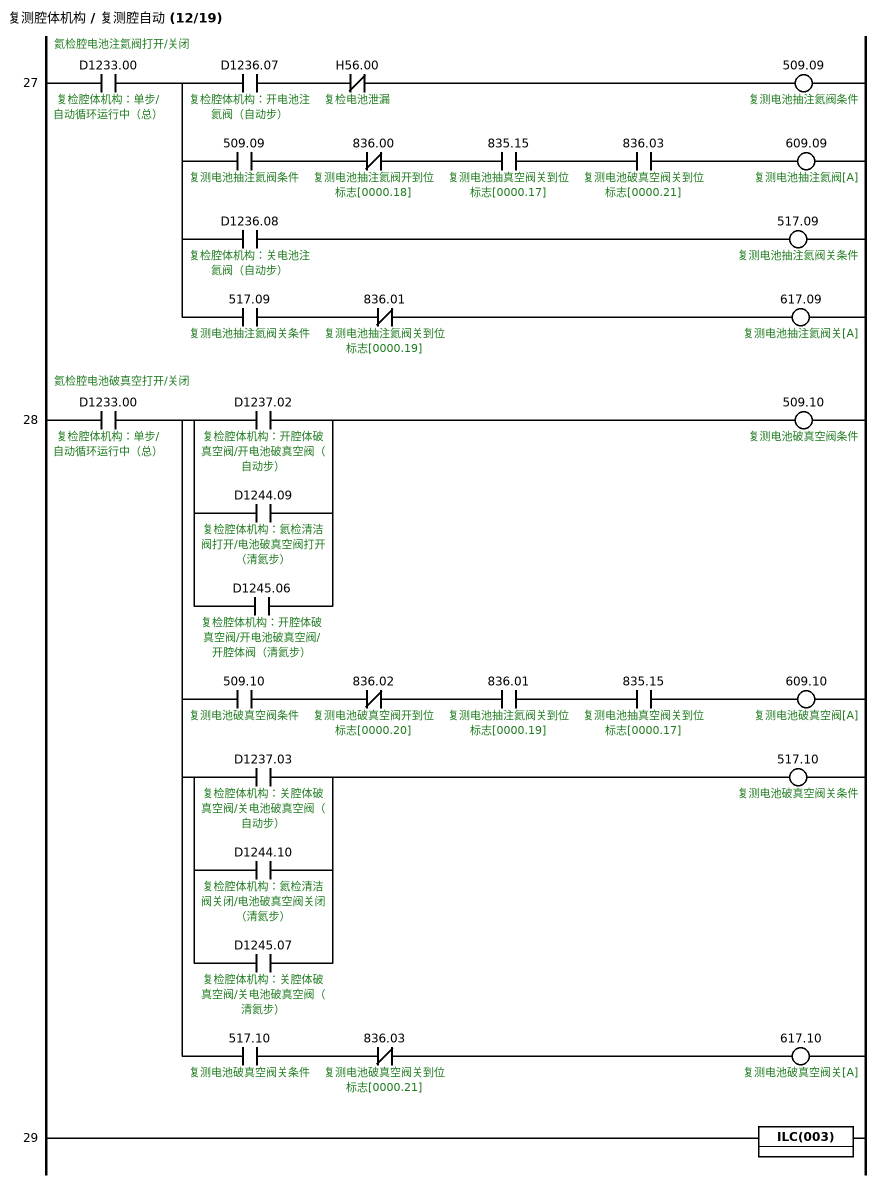
; [picture p600: 复测腔体机构 / 复测腔自动, rungs 27-29]
; rung 27: 氦检腔电池注氦阀打开/关闭
LD D1233.00  ; 复检腔体机构：单步/自动循环运行中（总）
OUT TR0
AND D1236.07  ; 复检腔体机构：开电池注氦阀（自动步）
ANDNOT H56.00  ; 复检电池泄漏
OUT 509.09  ; 复测电池抽注氦阀条件
LD TR0
AND 509.09  ; 复测电池抽注氦阀条件
ANDNOT 836.00  ; 复测电池抽注氦阀开到位标志[0000.18]
AND 835.15  ; 复测电池抽真空阀关到位标志[0000.17]
AND 836.03  ; 复测电池破真空阀关到位标志[0000.21]
OUT 609.09  ; 复测电池抽注氦阀[A]
LD TR0
AND D1236.08  ; 复检腔体机构：关电池注氦阀（自动步）
OUT 517.09  ; 复测电池抽注氦阀关条件
LD TR0
AND 517.09  ; 复测电池抽注氦阀关条件
ANDNOT 836.01  ; 复测电池抽注氦阀关到位标志[0000.19]
OUT 617.09  ; 复测电池抽注氦阀关[A]
; rung 28: 氦检腔电池破真空打开/关闭
LD D1233.00  ; 复检腔体机构：单步/自动循环运行中（总）
OUT TR0
LD D1237.02  ; 复检腔体机构：开腔体破真空阀/开电池破真空阀（自动步）
OR D1244.09  ; 复检腔体机构：氦检清洁阀打开/电池破真空阀打开（清氦步）
OR D1245.06  ; 复检腔体机构：开腔体破真空阀/开电池破真空阀/开腔体阀（清氦步）
ANDLD
OUT 509.10  ; 复测电池破真空阀条件
LD TR0
AND 509.10  ; 复测电池破真空阀条件
ANDNOT 836.02  ; 复测电池破真空阀开到位标志[0000.20]
AND 836.01  ; 复测电池抽注氦阀关到位标志[0000.19]
AND 835.15  ; 复测电池抽真空阀关到位标志[0000.17]
OUT 609.10  ; 复测电池破真空阀[A]
LD TR0
LD D1237.03  ; 复检腔体机构：关腔体破真空阀/关电池破真空阀（自动步）
OR D1244.10  ; 复检腔体机构：氦检清洁阀关闭/电池破真空阀关闭（清氦步）
OR D1245.07  ; 复检腔体机构：关腔体破真空阀/关电池破真空阀（清氦步）
ANDLD
OUT 517.10  ; 复测电池破真空阀关条件
LD TR0
AND 517.10  ; 复测电池破真空阀关条件
ANDNOT 836.03  ; 复测电池破真空阀关到位标志[0000.21]
OUT 617.10  ; 复测电池破真空阀关[A]
; rung 29
ILC(003)

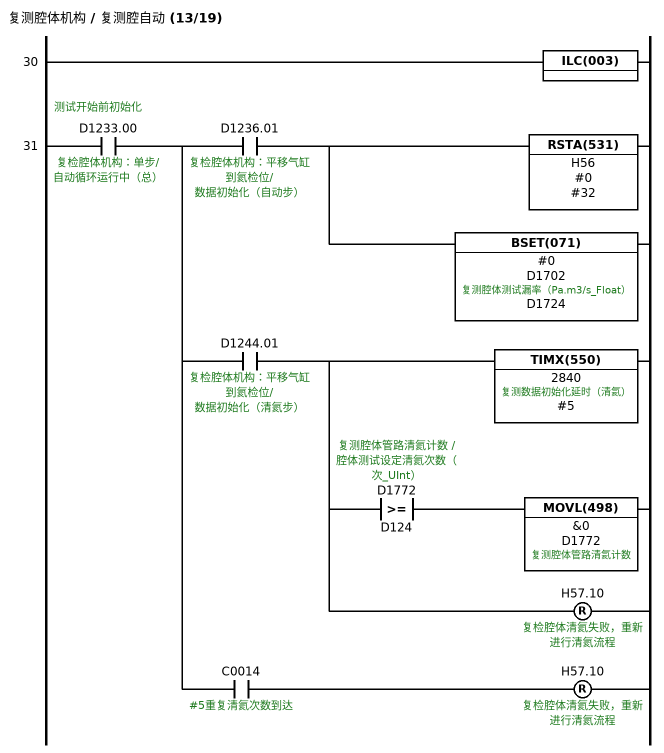
; rung 30
ILC(003)
; rung 31: 测试开始前初始化
LD D1233.00  ; 复检腔体机构：单步/自动循环运行中（总）
OUT TR0
AND D1236.01  ; 复检腔体机构：平移气缸到氦检位/数据初始化（自动步）
RSTA(531) H56 #0 #32
BSET(071) #0 D1702 D1724  ; 复测腔体测试漏率（Pa.m3/s_Float）
LD TR0
AND D1244.01  ; 复检腔体机构：平移气缸到氦检位/数据初始化（清氦步）
OUT TR1
TIMX(550) 2840 #5  ; 复测数据初始化延时（清氦）
AND>=(325) D1772 D124  ; 复测腔体管路清氦计数, 腔体测试设定清氦次数（次_UInt）
MOVL(498) &0 D1772  ; 复测腔体管路清氦计数
LD TR1
RSET H57.10  ; 复检腔体清氦失败，重新进行清氦流程
LD TR0
AND C0014  ; #5重复清氦次数到达
RSET H57.10  ; 复检腔体清氦失败，重新进行清氦流程

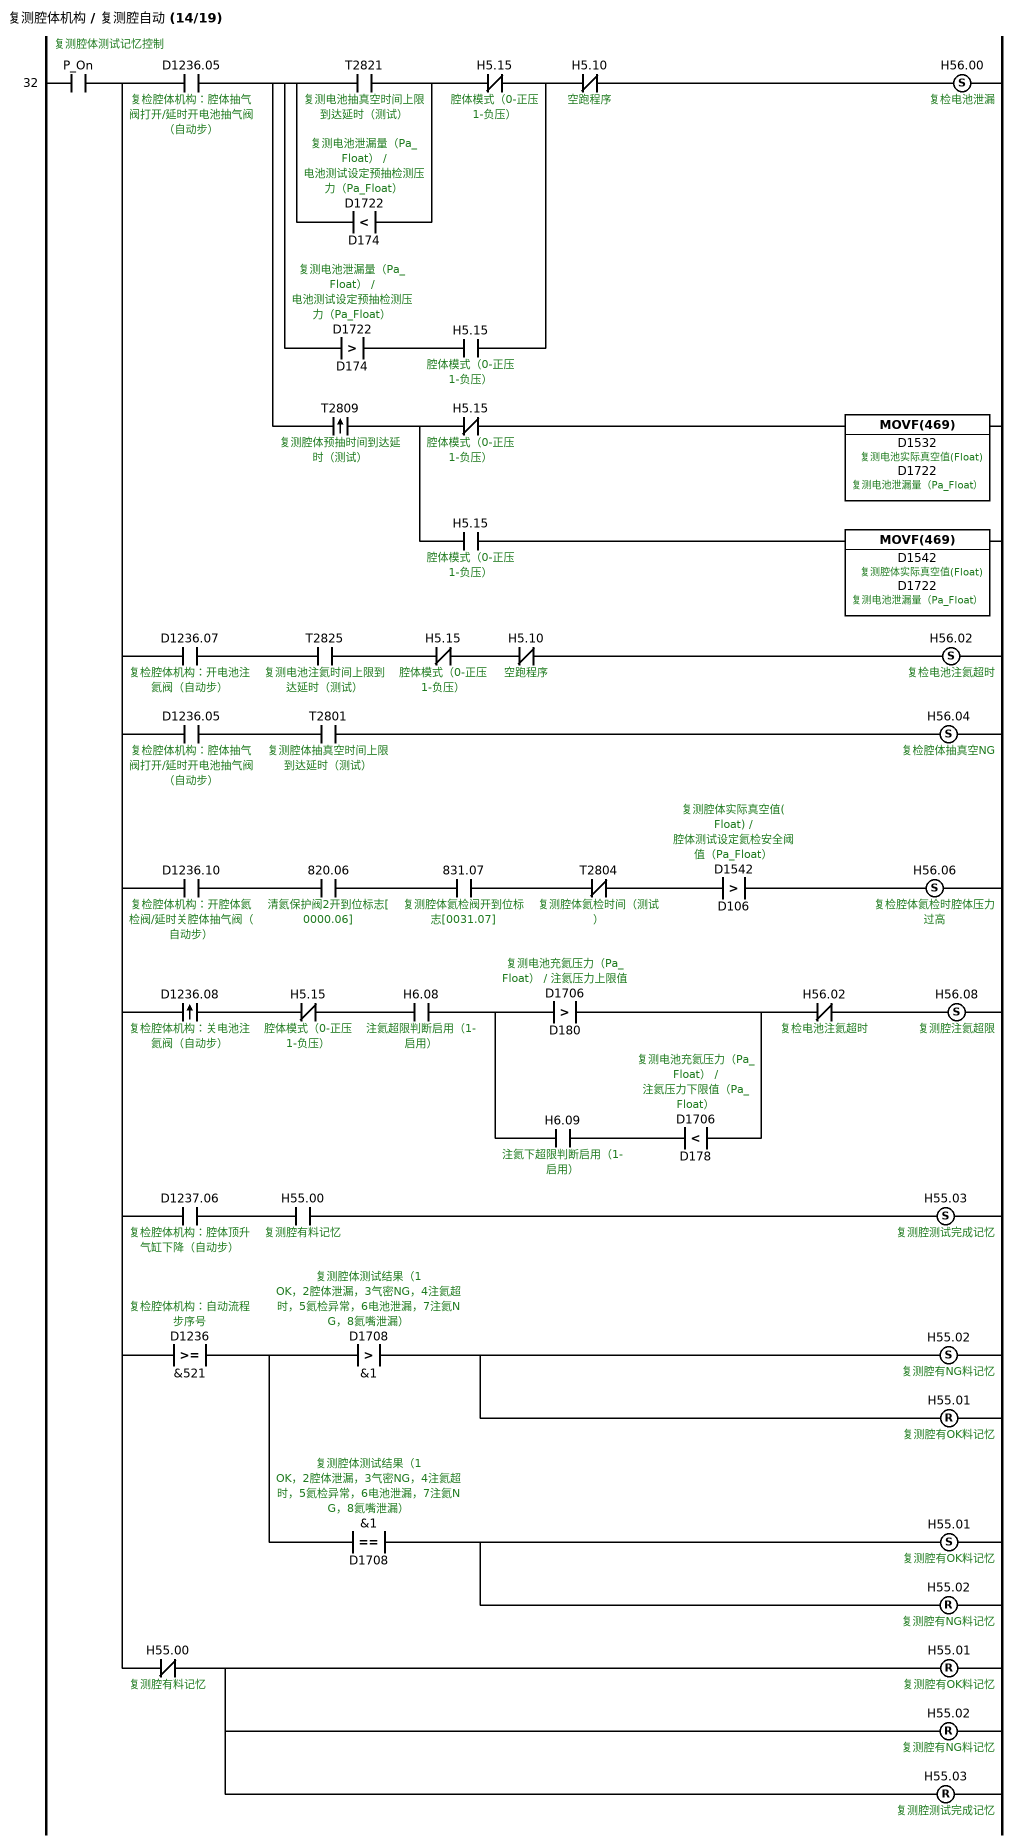
; rung 32: 复测腔体测试记忆控制
LD P_On
OUT TR0
AND D1236.05  ; 复检腔体机构：腔体抽气阀打开/延时开电池抽气阀（自动步）
OUT TR1
LD T2821  ; 复测电池抽真空时间上限到达延时（测试）
OR<F(331) D1722 D174  ; 复测电池泄漏量（Pa_Float）, 电池测试设定预抽检测压力（Pa_Float）
ANDNOT H5.15  ; 腔体模式（0-正压 1-负压）
LD>F(333) D1722 D174  ; 复测电池泄漏量（Pa_Float）, 电池测试设定预抽检测压力（Pa_Float）
AND H5.15  ; 腔体模式（0-正压 1-负压）
ORLD
ANDLD
ANDNOT H5.10  ; 空跑程序
SET H56.00  ; 复检电池泄漏
LD TR1
@AND T2809  ; 复测腔体预抽时间到达延时（测试）
OUT TR1
ANDNOT H5.15  ; 腔体模式（0-正压 1-负压）
MOVF(469) D1532 D1722  ; 复测电池实际真空值(Float), 复测电池泄漏量（Pa_Float）
LD TR1
AND H5.15  ; 腔体模式（0-正压 1-负压）
MOVF(469) D1542 D1722  ; 复测腔体实际真空值(Float), 复测电池泄漏量（Pa_Float）
LD TR0
AND D1236.07  ; 复检腔体机构：开电池注氦阀（自动步）
AND T2825  ; 复测电池注氦时间上限到达延时（测试）
ANDNOT H5.15  ; 腔体模式（0-正压 1-负压）
ANDNOT H5.10  ; 空跑程序
SET H56.02  ; 复检电池注氦超时
LD TR0
AND D1236.05  ; 复检腔体机构：腔体抽气阀打开/延时开电池抽气阀（自动步）
AND T2801  ; 复测腔体抽真空时间上限到达延时（测试）
SET H56.04  ; 复检腔体抽真空NG
LD TR0
AND D1236.10  ; 复检腔体机构：开腔体氦检阀/延时关腔体抽气阀（自动步）
AND 820.06  ; 清氦保护阀2开到位标志[0000.06]
AND 831.07  ; 复测腔体氦检阀开到位标志[0031.07]
ANDNOT T2804  ; 复测腔体氦检时间（测试）
AND>F(333) D1542 D106  ; 复测腔体实际真空值(Float), 腔体测试设定氦检安全阈值（Pa_Float）
SET H56.06  ; 复检腔体氦检时腔体压力过高
LD TR0
@AND D1236.08  ; 复检腔体机构：关电池注氦阀（自动步）
ANDNOT H5.15  ; 腔体模式（0-正压 1-负压）
AND H6.08  ; 注氦超限判断启用（1-启用）
LD>F(333) D1706 D180  ; 复测电池充氦压力（Pa_Float）, 注氦压力上限值
LD H6.09  ; 注氦下超限判断启用（1-启用）
AND<F(331) D1706 D178  ; 复测电池充氦压力（Pa_Float）, 注氦压力下限值（Pa_Float）
ORLD
ANDLD
ANDNOT H56.02  ; 复检电池注氦超时
SET H56.08  ; 复测腔注氦超限
LD TR0
AND D1237.06  ; 复检腔体机构：腔体顶升气缸下降（自动步）
AND H55.00  ; 复测腔有料记忆
SET H55.03  ; 复测腔测试完成记忆
LD TR0
AND>=L(326) D1236 &521  ; 复检腔体机构：自动流程步序号
OUT TR1
AND>(320) D1708 &1  ; 复测腔体测试结果（1 OK，2腔体泄漏，3气密NG，4注氦超时，5氦检异常，6电池泄漏，7注氦NG，8氦嘴泄漏）
SET H55.02  ; 复测腔有NG料记忆
RSET H55.01  ; 复测腔有OK料记忆
LD TR1
AND=(300) &1 D1708  ; 复测腔体测试结果（1 OK，2腔体泄漏，3气密NG，4注氦超时，5氦检异常，6电池泄漏，7注氦NG，8氦嘴泄漏）
SET H55.01  ; 复测腔有OK料记忆
RSET H55.02  ; 复测腔有NG料记忆
LD TR0
ANDNOT H55.00  ; 复测腔有料记忆
RSET H55.01  ; 复测腔有OK料记忆
RSET H55.02  ; 复测腔有NG料记忆
RSET H55.03  ; 复测腔测试完成记忆

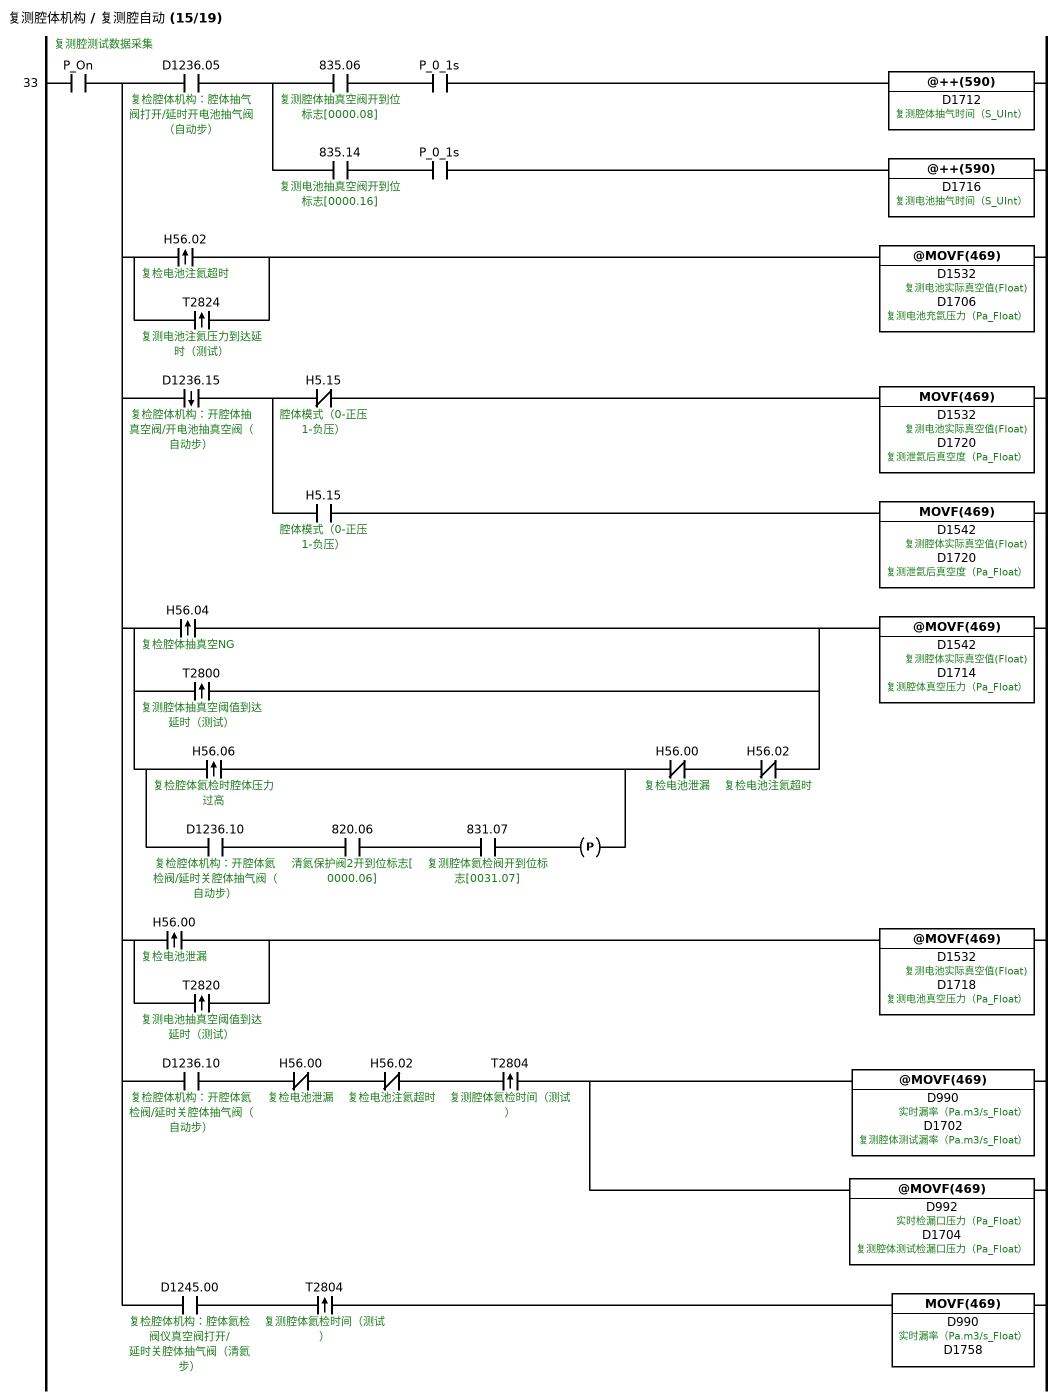
; rung 33: 复测腔测试数据采集
LD P_On
OUT TR0
AND D1236.05  ; 复检腔体机构：腔体抽气阀打开/延时开电池抽气阀（自动步）
OUT TR1
AND 835.06  ; 复测腔体抽真空阀开到位标志[0000.08]
AND P_0_1s
@++(590) D1712  ; 复测腔体抽气时间（S_UInt）
LD TR1
AND 835.14  ; 复测电池抽真空阀开到位标志[0000.16]
AND P_0_1s
@++(590) D1716  ; 复测电池抽气时间（S_UInt）
LD TR0
@LD H56.02  ; 复检电池注氦超时
@OR T2824  ; 复测电池注氦压力到达延时（测试）
ANDLD
@MOVF(469) D1532 D1706  ; 复测电池实际真空值(Float), 复测电池充氦压力（Pa_Float）
LD TR0
%AND D1236.15  ; 复检腔体机构：开腔体抽真空阀/开电池抽真空阀（自动步）
OUT TR1
ANDNOT H5.15  ; 腔体模式（0-正压 1-负压）
MOVF(469) D1532 D1720  ; 复测电池实际真空值(Float), 复测泄氦后真空度（Pa_Float）
LD TR1
AND H5.15  ; 腔体模式（0-正压 1-负压）
MOVF(469) D1542 D1720  ; 复测腔体实际真空值(Float), 复测泄氦后真空度（Pa_Float）
LD TR0
@LD H56.04  ; 复检腔体抽真空NG
@OR T2800  ; 复测腔体抽真空阈值到达延时（测试）
@LD H56.06  ; 复检腔体氦检时腔体压力过高
LD D1236.10  ; 复检腔体机构：开腔体氦检阀/延时关腔体抽气阀（自动步）
AND 820.06  ; 清氦保护阀2开到位标志[0000.06]
AND 831.07  ; 复测腔体氦检阀开到位标志[0031.07]
UP(521)
ORLD
ANDNOT H56.00  ; 复检电池泄漏
ANDNOT H56.02  ; 复检电池注氦超时
ORLD
ANDLD
@MOVF(469) D1542 D1714  ; 复测腔体实际真空值(Float), 复测腔体真空压力（Pa_Float）
LD TR0
@LD H56.00  ; 复检电池泄漏
@OR T2820  ; 复测电池抽真空阈值到达延时（测试）
ANDLD
@MOVF(469) D1532 D1718  ; 复测电池实际真空值(Float), 复测电池真空压力（Pa_Float）
LD TR0
AND D1236.10  ; 复检腔体机构：开腔体氦检阀/延时关腔体抽气阀（自动步）
ANDNOT H56.00  ; 复检电池泄漏
ANDNOT H56.02  ; 复检电池注氦超时
@AND T2804  ; 复测腔体氦检时间（测试）
@MOVF(469) D990 D1702  ; 实时漏率（Pa.m3/s_Float）, 复测腔体测试漏率（Pa.m3/s_Float）
@MOVF(469) D992 D1704  ; 实时检漏口压力（Pa_Float）, 复测腔体测试检漏口压力（Pa_Float）
LD TR0
AND D1245.00  ; 复检腔体机构：腔体氦检阀仪真空阀打开/延时关腔体抽气阀（清氦步）
@AND T2804  ; 复测腔体氦检时间（测试）
MOVF(469) D990 D1758  ; 实时漏率（Pa.m3/s_Float）

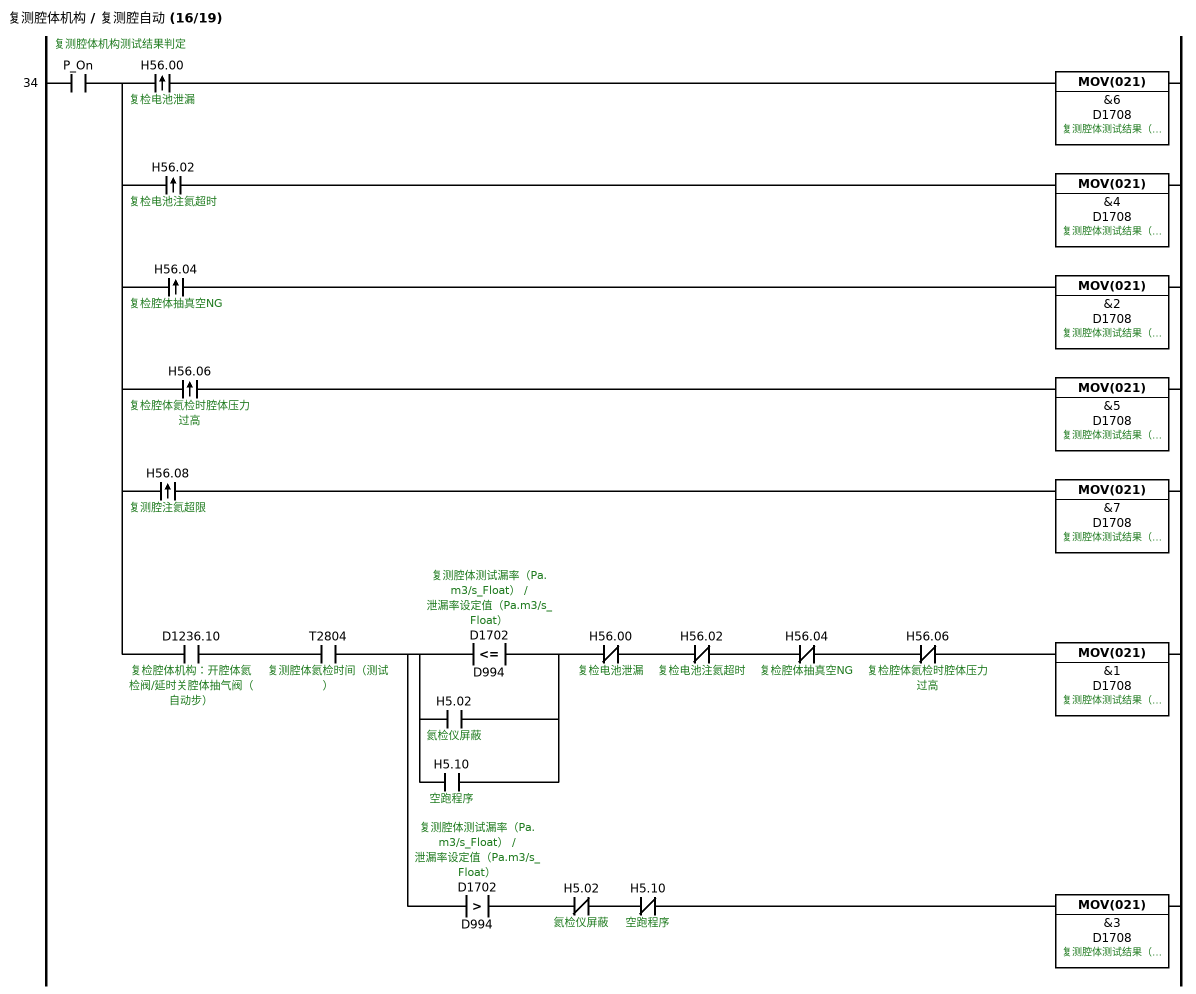
; rung 34: 复测腔体机构测试结果判定
LD P_On
OUT TR0
@AND H56.00  ; 复检电池泄漏
MOV(021) &6 D1708  ; 复测腔体测试结果（1 OK，2腔体泄漏，3气密NG，4注氦超时，5氦检异常，6电池泄漏，7注氦NG，8氦嘴泄漏）
LD TR0
@AND H56.02  ; 复检电池注氦超时
MOV(021) &4 D1708  ; 复测腔体测试结果（1 OK，2腔体泄漏，3气密NG，4注氦超时，5氦检异常，6电池泄漏，7注氦NG，8氦嘴泄漏）
LD TR0
@AND H56.04  ; 复检腔体抽真空NG
MOV(021) &2 D1708  ; 复测腔体测试结果（1 OK，2腔体泄漏，3气密NG，4注氦超时，5氦检异常，6电池泄漏，7注氦NG，8氦嘴泄漏）
LD TR0
@AND H56.06  ; 复检腔体氦检时腔体压力过高
MOV(021) &5 D1708  ; 复测腔体测试结果（1 OK，2腔体泄漏，3气密NG，4注氦超时，5氦检异常，6电池泄漏，7注氦NG，8氦嘴泄漏）
LD TR0
@AND H56.08  ; 复测腔注氦超限
MOV(021) &7 D1708  ; 复测腔体测试结果（1 OK，2腔体泄漏，3气密NG，4注氦超时，5氦检异常，6电池泄漏，7注氦NG，8氦嘴泄漏）
LD TR0
AND D1236.10  ; 复检腔体机构：开腔体氦检阀/延时关腔体抽气阀（自动步）
AND T2804  ; 复测腔体氦检时间（测试）
OUT TR0
LD<=F(332) D1702 D994  ; 复测腔体测试漏率（Pa.m3/s_Float）, 泄漏率设定值（Pa.m3/s_Float）
OR H5.02  ; 氦检仪屏蔽
OR H5.10  ; 空跑程序
ANDLD
ANDNOT H56.00  ; 复检电池泄漏
ANDNOT H56.02  ; 复检电池注氦超时
ANDNOT H56.04  ; 复检腔体抽真空NG
ANDNOT H56.06  ; 复检腔体氦检时腔体压力过高
MOV(021) &1 D1708  ; 复测腔体测试结果（1 OK，2腔体泄漏，3气密NG，4注氦超时，5氦检异常，6电池泄漏，7注氦NG，8氦嘴泄漏）
LD TR0
AND>F(333) D1702 D994  ; 复测腔体测试漏率（Pa.m3/s_Float）, 泄漏率设定值（Pa.m3/s_Float）
ANDNOT H5.02  ; 氦检仪屏蔽
ANDNOT H5.10  ; 空跑程序
MOV(021) &3 D1708  ; 复测腔体测试结果（1 OK，2腔体泄漏，3气密NG，4注氦超时，5氦检异常，6电池泄漏，7注氦NG，8氦嘴泄漏）

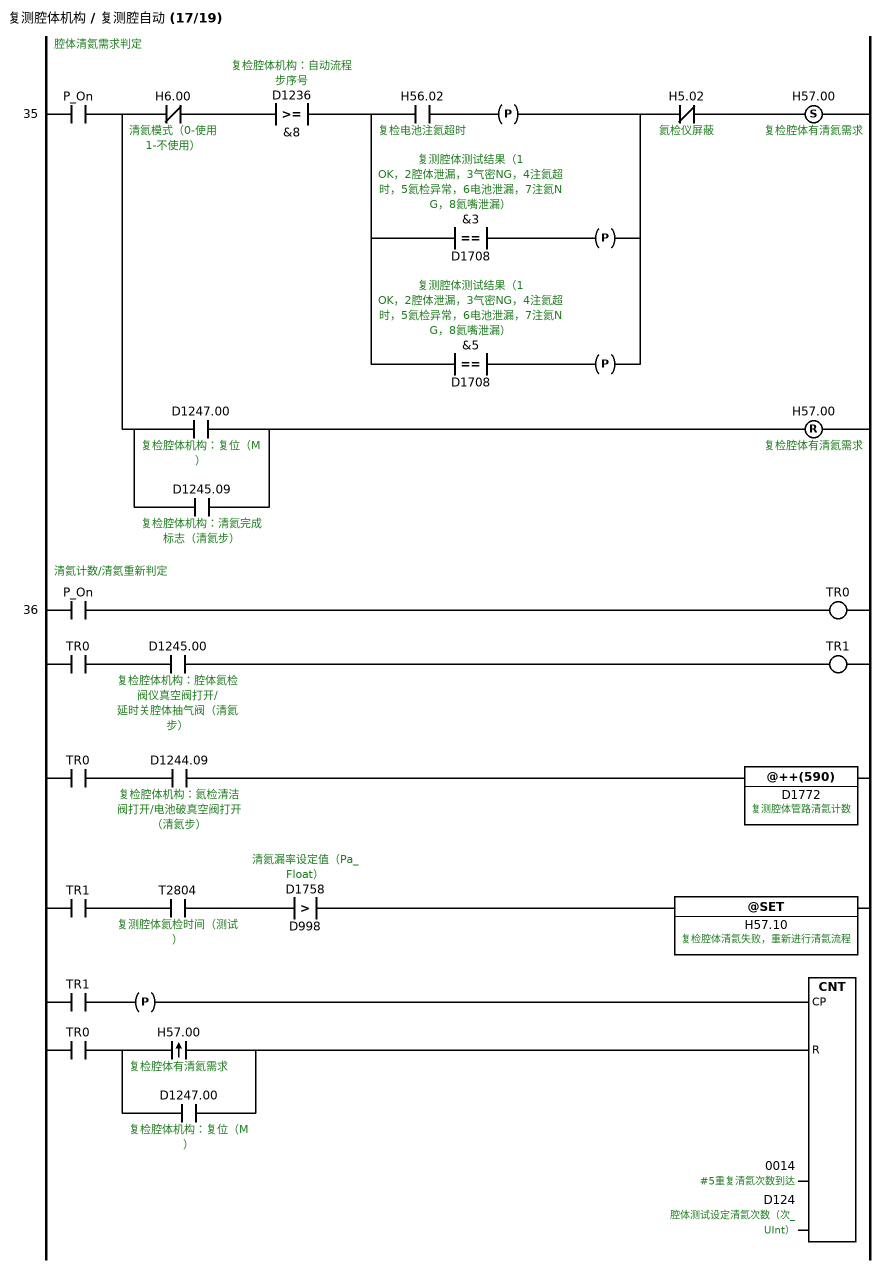
; rung 35: 腔体清氦需求判定
LD P_On
OUT TR0
ANDNOT H6.00  ; 清氦模式（0-使用 1-不使用）
AND>=L(326) D1236 &8  ; 复检腔体机构：自动流程步序号
LD H56.02  ; 复检电池注氦超时
UP(521)
LD=(300) &3 D1708  ; 复测腔体测试结果（1 OK，2腔体泄漏，3气密NG，4注氦超时，5氦检异常，6电池泄漏，7注氦NG，8氦嘴泄漏）
UP(521)
ORLD
LD=(300) &5 D1708  ; 复测腔体测试结果（1 OK，2腔体泄漏，3气密NG，4注氦超时，5氦检异常，6电池泄漏，7注氦NG，8氦嘴泄漏）
UP(521)
ORLD
ANDLD
ANDNOT H5.02  ; 氦检仪屏蔽
SET H57.00  ; 复检腔体有清氦需求
LD TR0
LD D1247.00  ; 复检腔体机构：复位（M）
OR D1245.09  ; 复检腔体机构：清氦完成标志（清氦步）
ANDLD
RSET H57.00  ; 复检腔体有清氦需求
; rung 36: 清氦计数/清氦重新判定
LD P_On
OUT TR0
AND D1244.09  ; 复检腔体机构：氦检清洁阀打开/电池破真空阀打开（清氦步）
@++(590) D1772  ; 复测腔体管路清氦计数
LD TR0
AND D1245.00  ; 复检腔体机构：腔体氦检阀仪真空阀打开/延时关腔体抽气阀（清氦步）
OUT TR1
AND T2804  ; 复测腔体氦检时间（测试）
AND>F(333) D1758 D998  ; 清氦漏率设定值（Pa_Float）
@SET H57.10  ; 复检腔体清氦失败，重新进行清氦流程
LD TR1
UP(521)
LD TR0
@LD H57.00  ; 复检腔体有清氦需求
OR D1247.00  ; 复检腔体机构：复位（M）
ANDLD
CNT 0014 D124  ; 腔体测试设定清氦次数（次_UInt）, #5重复清氦次数到达

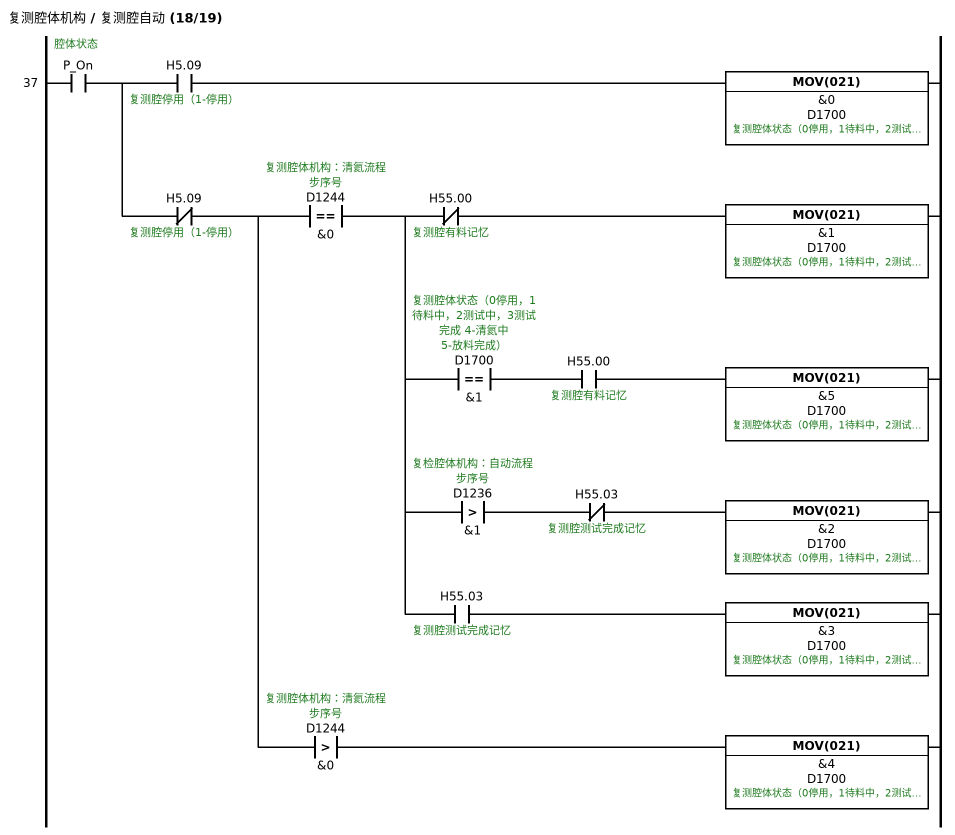
; rung 37: 腔体状态
LD P_On
OUT TR0
AND H5.09  ; 复测腔停用（1-停用）
MOV(021) &0 D1700  ; 复测腔体状态（0停用，1待料中，2测试中，3测试完成 4-清氦中  5-放料完成）
LD TR0
ANDNOT H5.09  ; 复测腔停用（1-停用）
OUT TR0
AND=L(301) D1244 &0  ; 复测腔体机构：清氦流程步序号
OUT TR1
ANDNOT H55.00  ; 复测腔有料记忆
MOV(021) &1 D1700  ; 复测腔体状态（0停用，1待料中，2测试中，3测试完成 4-清氦中  5-放料完成）
LD TR1
AND=(300) D1700 &1  ; 复测腔体状态（0停用，1待料中，2测试中，3测试完成 4-清氦中  5-放料完成）
AND H55.00  ; 复测腔有料记忆
MOV(021) &5 D1700  ; 复测腔体状态（0停用，1待料中，2测试中，3测试完成 4-清氦中  5-放料完成）
LD TR1
AND>L(321) D1236 &1  ; 复检腔体机构：自动流程步序号
ANDNOT H55.03  ; 复测腔测试完成记忆
MOV(021) &2 D1700  ; 复测腔体状态（0停用，1待料中，2测试中，3测试完成 4-清氦中  5-放料完成）
LD TR1
AND H55.03  ; 复测腔测试完成记忆
MOV(021) &3 D1700  ; 复测腔体状态（0停用，1待料中，2测试中，3测试完成 4-清氦中  5-放料完成）
LD TR0
AND>L(321) D1244 &0  ; 复测腔体机构：清氦流程步序号
MOV(021) &4 D1700  ; 复测腔体状态（0停用，1待料中，2测试中，3测试完成 4-清氦中  5-放料完成）

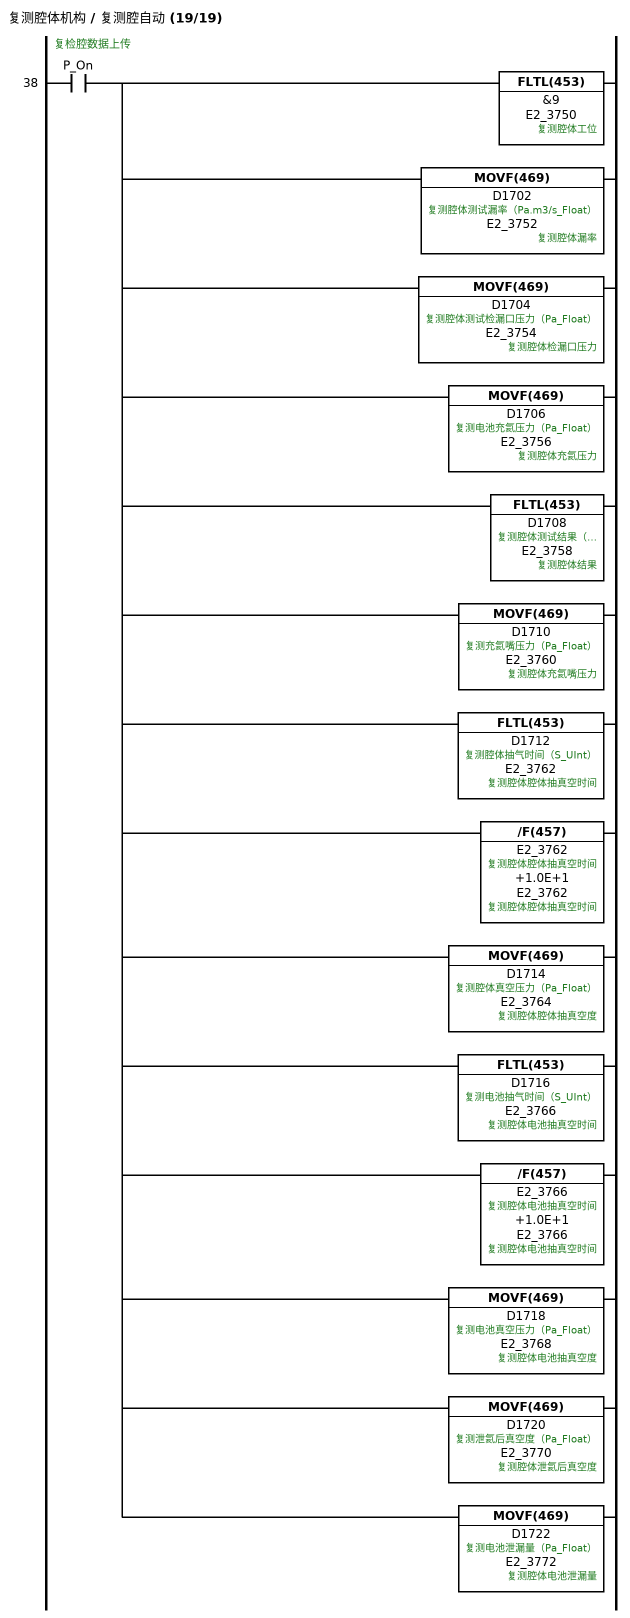
; rung 38: 复检腔数据上传
LD P_On
FLTL(453) &9 E2_3750  ; 复测腔体工位
MOVF(469) D1702 E2_3752  ; 复测腔体测试漏率（Pa.m3/s_Float）, 复测腔体漏率
MOVF(469) D1704 E2_3754  ; 复测腔体测试检漏口压力（Pa_Float）, 复测腔体检漏口压力
MOVF(469) D1706 E2_3756  ; 复测电池充氦压力（Pa_Float）, 复测腔体充氦压力
FLTL(453) D1708 E2_3758  ; 复测腔体测试结果（1 OK，2腔体泄漏，3气密NG，4注氦超时，5氦检异常，6电池泄漏，7注氦NG，8氦嘴泄漏）, 复测腔体结果
MOVF(469) D1710 E2_3760  ; 复测充氦嘴压力（Pa_Float）, 复测腔体充氦嘴压力
FLTL(453) D1712 E2_3762  ; 复测腔体抽气时间（S_UInt）, 复测腔体腔体抽真空时间
/F(457) E2_3762 +1.0E+1 E2_3762  ; 复测腔体腔体抽真空时间
MOVF(469) D1714 E2_3764  ; 复测腔体真空压力（Pa_Float）, 复测腔体腔体抽真空度
FLTL(453) D1716 E2_3766  ; 复测电池抽气时间（S_UInt）, 复测腔体电池抽真空时间
/F(457) E2_3766 +1.0E+1 E2_3766  ; 复测腔体电池抽真空时间
MOVF(469) D1718 E2_3768  ; 复测电池真空压力（Pa_Float）, 复测腔体电池抽真空度
MOVF(469) D1720 E2_3770  ; 复测泄氦后真空度（Pa_Float）, 复测腔体泄氦后真空度
MOVF(469) D1722 E2_3772  ; 复测电池泄漏量（Pa_Float）, 复测腔体电池泄漏量

### Section 复测腔手动

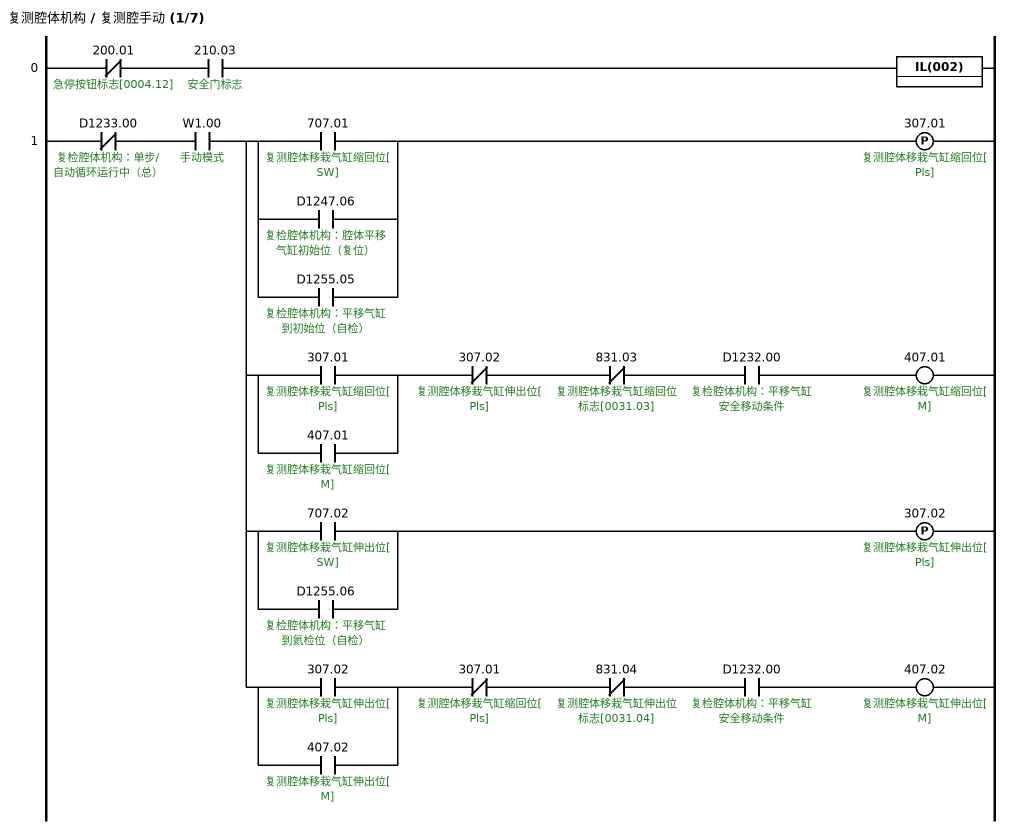
; rung 0
LDNOT 200.01  ; 急停按钮标志[0004.12]
AND 210.03  ; 安全门标志
IL(002)
; rung 1
LDNOT D1233.00  ; 复检腔体机构：单步/自动循环运行中（总）
AND W1.00  ; 手动模式
OUT TR0
LD 707.01  ; 复测腔体移栽气缸缩回位[SW]
OR D1247.06  ; 复检腔体机构：腔体平移气缸初始位（复位）
OR D1255.05  ; 复检腔体机构：平移气缸到初始位（自检）
ANDLD
DIFU(013) 307.01  ; 复测腔体移栽气缸缩回位[Pls]
LD TR0
LD 307.01  ; 复测腔体移栽气缸缩回位[Pls]
OR 407.01  ; 复测腔体移栽气缸缩回位[M]
ANDLD
ANDNOT 307.02  ; 复测腔体移栽气缸伸出位[Pls]
ANDNOT 831.03  ; 复测腔体移栽气缸缩回位标志[0031.03]
AND D1232.00  ; 复检腔体机构：平移气缸安全移动条件
OUT 407.01  ; 复测腔体移栽气缸缩回位[M]
LD TR0
LD 707.02  ; 复测腔体移栽气缸伸出位[SW]
OR D1255.06  ; 复检腔体机构：平移气缸到氦检位（自检）
ANDLD
DIFU(013) 307.02  ; 复测腔体移栽气缸伸出位[Pls]
LD TR0
LD 307.02  ; 复测腔体移栽气缸伸出位[Pls]
OR 407.02  ; 复测腔体移栽气缸伸出位[M]
ANDLD
ANDNOT 307.01  ; 复测腔体移栽气缸缩回位[Pls]
ANDNOT 831.04  ; 复测腔体移栽气缸伸出位标志[0031.04]
AND D1232.00  ; 复检腔体机构：平移气缸安全移动条件
OUT 407.02  ; 复测腔体移栽气缸伸出位[M]

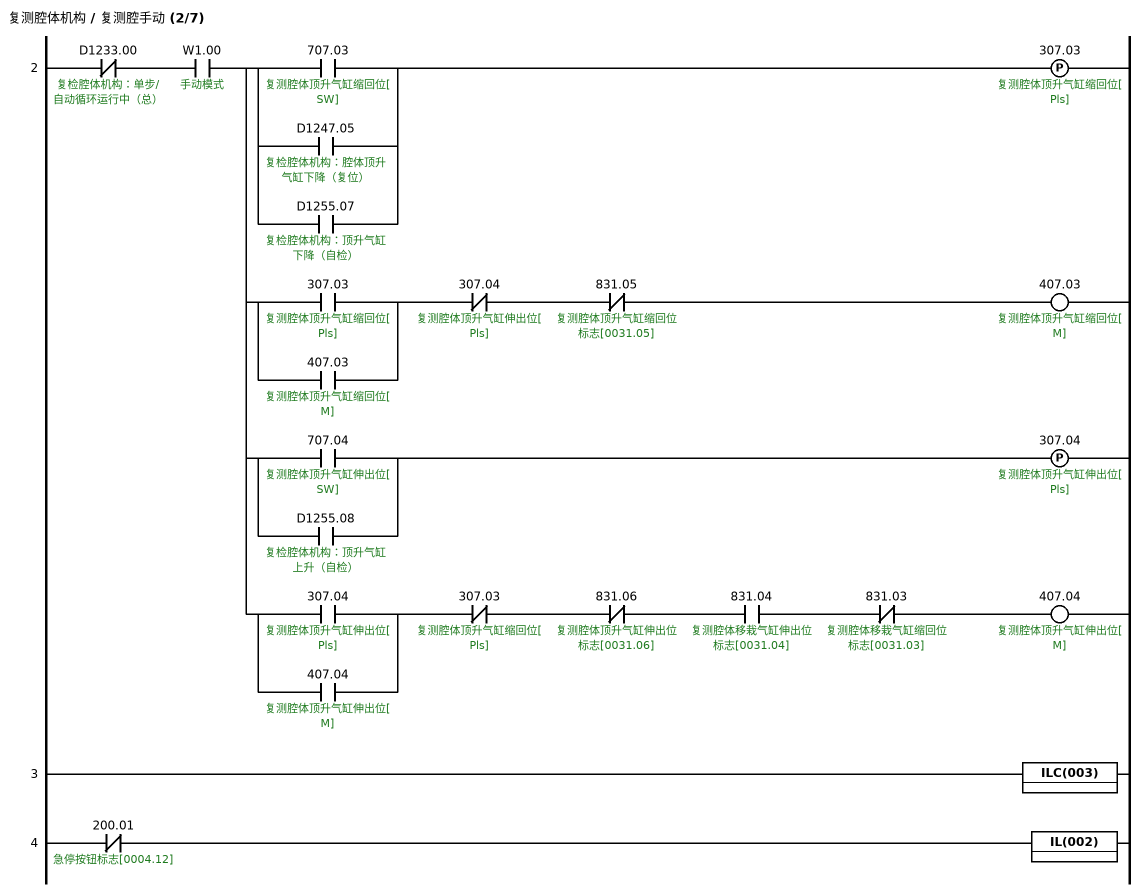
; rung 2
LDNOT D1233.00  ; 复检腔体机构：单步/自动循环运行中（总）
AND W1.00  ; 手动模式
OUT TR0
LD 707.03  ; 复测腔体顶升气缸缩回位[SW]
OR D1247.05  ; 复检腔体机构：腔体顶升气缸下降（复位）
OR D1255.07  ; 复检腔体机构：顶升气缸下降（自检）
ANDLD
DIFU(013) 307.03  ; 复测腔体顶升气缸缩回位[Pls]
LD TR0
LD 307.03  ; 复测腔体顶升气缸缩回位[Pls]
OR 407.03  ; 复测腔体顶升气缸缩回位[M]
ANDLD
ANDNOT 307.04  ; 复测腔体顶升气缸伸出位[Pls]
ANDNOT 831.05  ; 复测腔体顶升气缸缩回位标志[0031.05]
OUT 407.03  ; 复测腔体顶升气缸缩回位[M]
LD TR0
LD 707.04  ; 复测腔体顶升气缸伸出位[SW]
OR D1255.08  ; 复检腔体机构：顶升气缸上升（自检）
ANDLD
DIFU(013) 307.04  ; 复测腔体顶升气缸伸出位[Pls]
LD TR0
LD 307.04  ; 复测腔体顶升气缸伸出位[Pls]
OR 407.04  ; 复测腔体顶升气缸伸出位[M]
ANDLD
ANDNOT 307.03  ; 复测腔体顶升气缸缩回位[Pls]
ANDNOT 831.06  ; 复测腔体顶升气缸伸出位标志[0031.06]
AND 831.04  ; 复测腔体移栽气缸伸出位标志[0031.04]
ANDNOT 831.03  ; 复测腔体移栽气缸缩回位标志[0031.03]
OUT 407.04  ; 复测腔体顶升气缸伸出位[M]
; rung 3
ILC(003)
; rung 4
LDNOT 200.01  ; 急停按钮标志[0004.12]
IL(002)

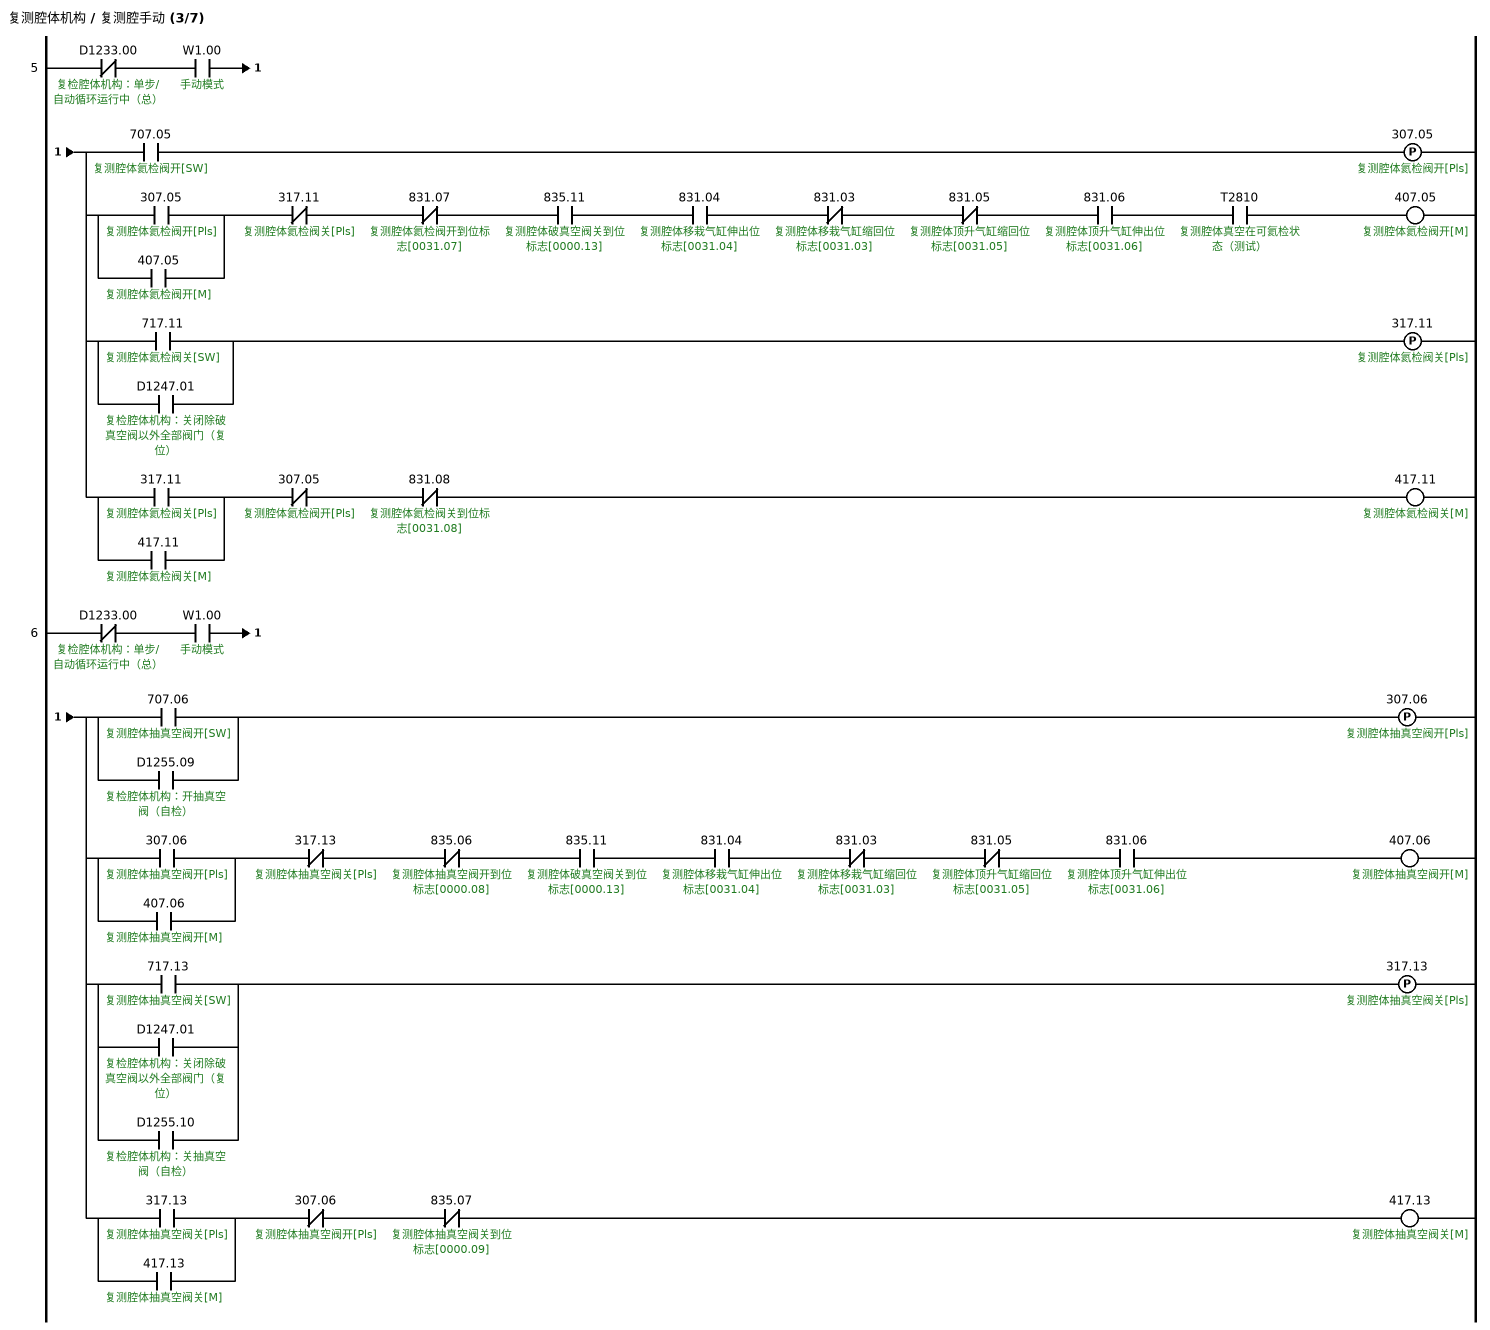
; rung 5
LDNOT D1233.00  ; 复检腔体机构：单步/自动循环运行中（总）
AND W1.00  ; 手动模式
OUT TR0
AND 707.05  ; 复测腔体氦检阀开[SW]
DIFU(013) 307.05  ; 复测腔体氦检阀开[Pls]
LD TR0
LD 307.05  ; 复测腔体氦检阀开[Pls]
OR 407.05  ; 复测腔体氦检阀开[M]
ANDLD
ANDNOT 317.11  ; 复测腔体氦检阀关[Pls]
ANDNOT 831.07  ; 复测腔体氦检阀开到位标志[0031.07]
AND 835.11  ; 复测腔体破真空阀关到位标志[0000.13]
AND 831.04  ; 复测腔体移栽气缸伸出位标志[0031.04]
ANDNOT 831.03  ; 复测腔体移栽气缸缩回位标志[0031.03]
ANDNOT 831.05  ; 复测腔体顶升气缸缩回位标志[0031.05]
AND 831.06  ; 复测腔体顶升气缸伸出位标志[0031.06]
AND T2810  ; 复测腔体真空在可氦检状态（测试）
OUT 407.05  ; 复测腔体氦检阀开[M]
LD TR0
LD 717.11  ; 复测腔体氦检阀关[SW]
OR D1247.01  ; 复检腔体机构：关闭除破真空阀以外全部阀门（复位）
ANDLD
DIFU(013) 317.11  ; 复测腔体氦检阀关[Pls]
LD TR0
LD 317.11  ; 复测腔体氦检阀关[Pls]
OR 417.11  ; 复测腔体氦检阀关[M]
ANDLD
ANDNOT 307.05  ; 复测腔体氦检阀开[Pls]
ANDNOT 831.08  ; 复测腔体氦检阀关到位标志[0031.08]
OUT 417.11  ; 复测腔体氦检阀关[M]
; rung 6
LDNOT D1233.00  ; 复检腔体机构：单步/自动循环运行中（总）
AND W1.00  ; 手动模式
OUT TR0
LD 707.06  ; 复测腔体抽真空阀开[SW]
OR D1255.09  ; 复检腔体机构：开抽真空阀（自检）
ANDLD
DIFU(013) 307.06  ; 复测腔体抽真空阀开[Pls]
LD TR0
LD 307.06  ; 复测腔体抽真空阀开[Pls]
OR 407.06  ; 复测腔体抽真空阀开[M]
ANDLD
ANDNOT 317.13  ; 复测腔体抽真空阀关[Pls]
ANDNOT 835.06  ; 复测腔体抽真空阀开到位标志[0000.08]
AND 835.11  ; 复测腔体破真空阀关到位标志[0000.13]
AND 831.04  ; 复测腔体移栽气缸伸出位标志[0031.04]
ANDNOT 831.03  ; 复测腔体移栽气缸缩回位标志[0031.03]
ANDNOT 831.05  ; 复测腔体顶升气缸缩回位标志[0031.05]
AND 831.06  ; 复测腔体顶升气缸伸出位标志[0031.06]
OUT 407.06  ; 复测腔体抽真空阀开[M]
LD TR0
LD 717.13  ; 复测腔体抽真空阀关[SW]
OR D1247.01  ; 复检腔体机构：关闭除破真空阀以外全部阀门（复位）
OR D1255.10  ; 复检腔体机构：关抽真空阀（自检）
ANDLD
DIFU(013) 317.13  ; 复测腔体抽真空阀关[Pls]
LD TR0
LD 317.13  ; 复测腔体抽真空阀关[Pls]
OR 417.13  ; 复测腔体抽真空阀关[M]
ANDLD
ANDNOT 307.06  ; 复测腔体抽真空阀开[Pls]
ANDNOT 835.07  ; 复测腔体抽真空阀关到位标志[0000.09]
OUT 417.13  ; 复测腔体抽真空阀关[M]

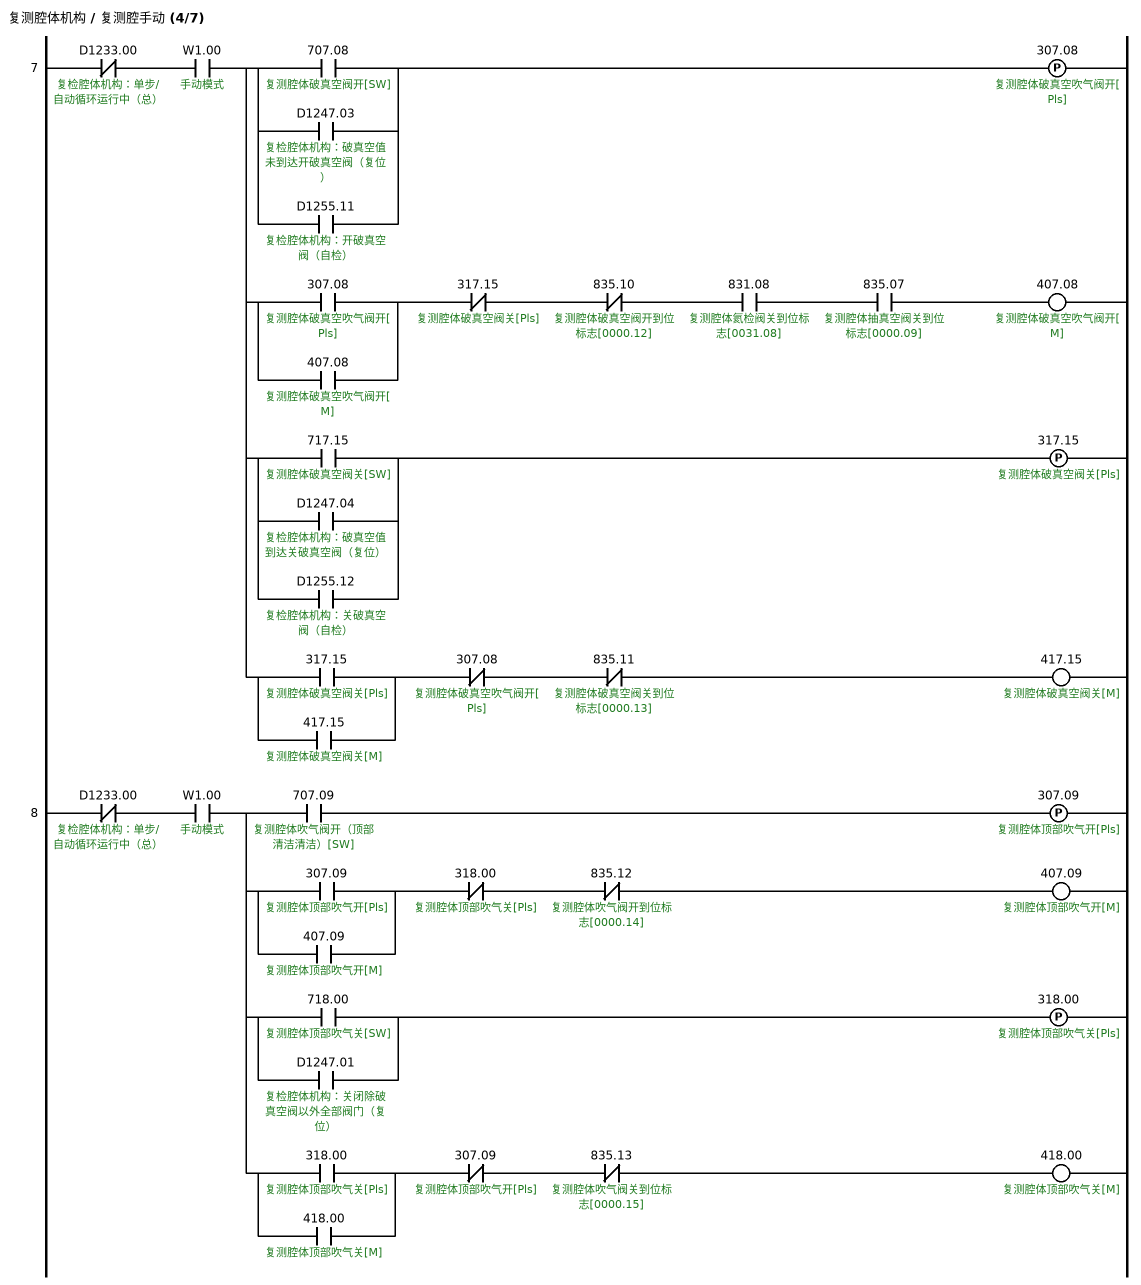
; rung 7
LDNOT D1233.00  ; 复检腔体机构：单步/自动循环运行中（总）
AND W1.00  ; 手动模式
OUT TR0
LD 707.08  ; 复测腔体破真空阀开[SW]
OR D1247.03  ; 复检腔体机构：破真空值未到达开破真空阀（复位）
OR D1255.11  ; 复检腔体机构：开破真空阀（自检）
ANDLD
DIFU(013) 307.08  ; 复测腔体破真空吹气阀开[Pls]
LD TR0
LD 307.08  ; 复测腔体破真空吹气阀开[Pls]
OR 407.08  ; 复测腔体破真空吹气阀开[M]
ANDLD
ANDNOT 317.15  ; 复测腔体破真空阀关[Pls]
ANDNOT 835.10  ; 复测腔体破真空阀开到位标志[0000.12]
AND 831.08  ; 复测腔体氦检阀关到位标志[0031.08]
AND 835.07  ; 复测腔体抽真空阀关到位标志[0000.09]
OUT 407.08  ; 复测腔体破真空吹气阀开[M]
LD TR0
LD 717.15  ; 复测腔体破真空阀关[SW]
OR D1247.04  ; 复检腔体机构：破真空值到达关破真空阀（复位）
OR D1255.12  ; 复检腔体机构：关破真空阀（自检）
ANDLD
DIFU(013) 317.15  ; 复测腔体破真空阀关[Pls]
LD TR0
LD 317.15  ; 复测腔体破真空阀关[Pls]
OR 417.15  ; 复测腔体破真空阀关[M]
ANDLD
ANDNOT 307.08  ; 复测腔体破真空吹气阀开[Pls]
ANDNOT 835.11  ; 复测腔体破真空阀关到位标志[0000.13]
OUT 417.15  ; 复测腔体破真空阀关[M]
; rung 8
LDNOT D1233.00  ; 复检腔体机构：单步/自动循环运行中（总）
AND W1.00  ; 手动模式
OUT TR0
AND 707.09  ; 复测腔体吹气阀开（顶部清洁清洁）[SW]
DIFU(013) 307.09  ; 复测腔体顶部吹气开[Pls]
LD TR0
LD 307.09  ; 复测腔体顶部吹气开[Pls]
OR 407.09  ; 复测腔体顶部吹气开[M]
ANDLD
ANDNOT 318.00  ; 复测腔体顶部吹气关[Pls]
ANDNOT 835.12  ; 复测腔体吹气阀开到位标志[0000.14]
OUT 407.09  ; 复测腔体顶部吹气开[M]
LD TR0
LD 718.00  ; 复测腔体顶部吹气关[SW]
OR D1247.01  ; 复检腔体机构：关闭除破真空阀以外全部阀门（复位）
ANDLD
DIFU(013) 318.00  ; 复测腔体顶部吹气关[Pls]
LD TR0
LD 318.00  ; 复测腔体顶部吹气关[Pls]
OR 418.00  ; 复测腔体顶部吹气关[M]
ANDLD
ANDNOT 307.09  ; 复测腔体顶部吹气开[Pls]
ANDNOT 835.13  ; 复测腔体吹气阀关到位标志[0000.15]
OUT 418.00  ; 复测腔体顶部吹气关[M]

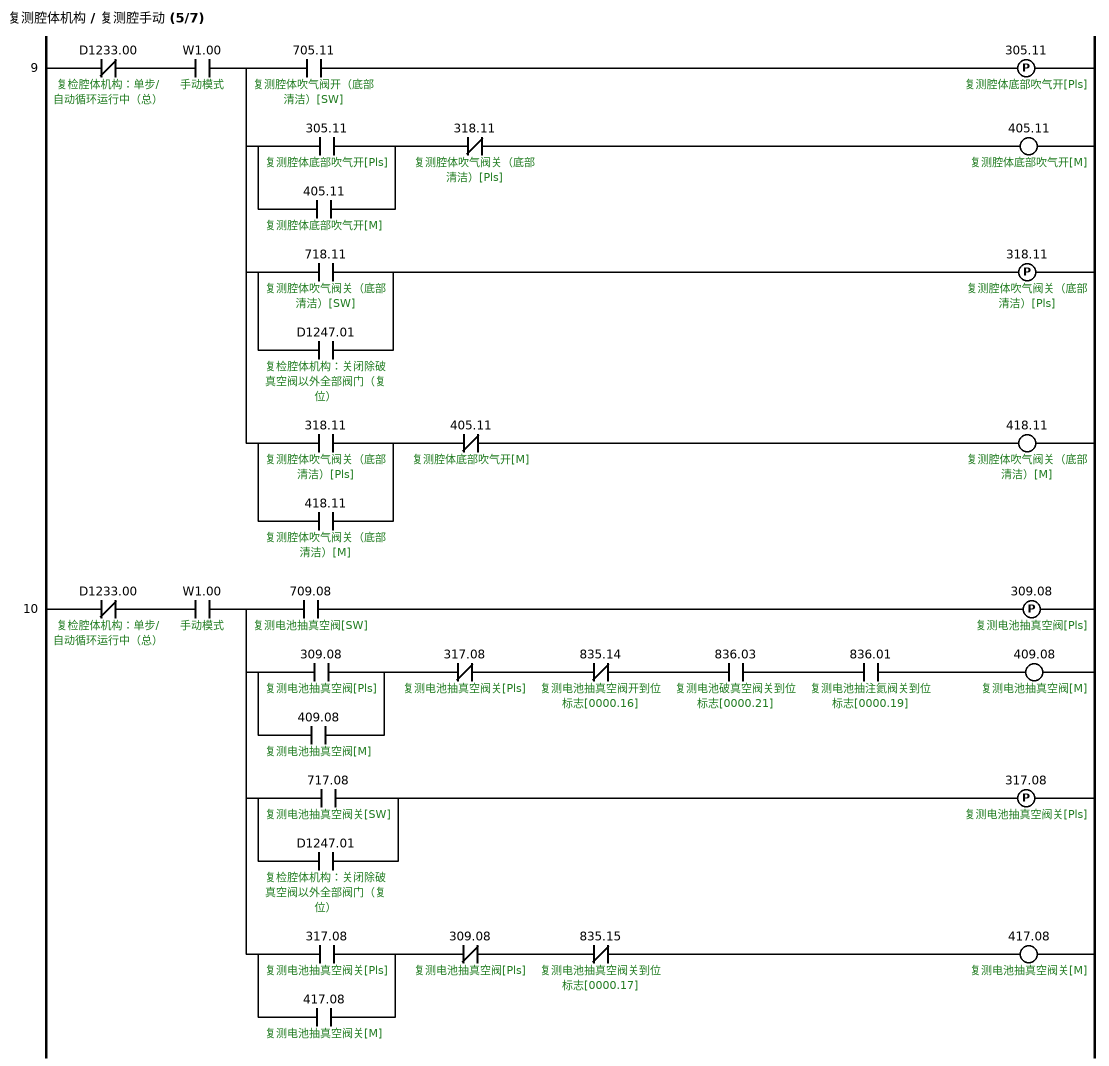
; rung 9
LDNOT D1233.00  ; 复检腔体机构：单步/自动循环运行中（总）
AND W1.00  ; 手动模式
OUT TR0
AND 705.11  ; 复测腔体吹气阀开（底部清洁）[SW]
DIFU(013) 305.11  ; 复测腔体底部吹气开[Pls]
LD TR0
LD 305.11  ; 复测腔体底部吹气开[Pls]
OR 405.11  ; 复测腔体底部吹气开[M]
ANDLD
ANDNOT 318.11  ; 复测腔体吹气阀关（底部清洁）[Pls]
OUT 405.11  ; 复测腔体底部吹气开[M]
LD TR0
LD 718.11  ; 复测腔体吹气阀关（底部清洁）[SW]
OR D1247.01  ; 复检腔体机构：关闭除破真空阀以外全部阀门（复位）
ANDLD
DIFU(013) 318.11  ; 复测腔体吹气阀关（底部清洁）[Pls]
LD TR0
LD 318.11  ; 复测腔体吹气阀关（底部清洁）[Pls]
OR 418.11  ; 复测腔体吹气阀关（底部清洁）[M]
ANDLD
ANDNOT 405.11  ; 复测腔体底部吹气开[M]
OUT 418.11  ; 复测腔体吹气阀关（底部清洁）[M]
; rung 10
LDNOT D1233.00  ; 复检腔体机构：单步/自动循环运行中（总）
AND W1.00  ; 手动模式
OUT TR0
AND 709.08  ; 复测电池抽真空阀[SW]
DIFU(013) 309.08  ; 复测电池抽真空阀[Pls]
LD TR0
LD 309.08  ; 复测电池抽真空阀[Pls]
OR 409.08  ; 复测电池抽真空阀[M]
ANDLD
ANDNOT 317.08  ; 复测电池抽真空阀关[Pls]
ANDNOT 835.14  ; 复测电池抽真空阀开到位标志[0000.16]
AND 836.03  ; 复测电池破真空阀关到位标志[0000.21]
AND 836.01  ; 复测电池抽注氦阀关到位标志[0000.19]
OUT 409.08  ; 复测电池抽真空阀[M]
LD TR0
LD 717.08  ; 复测电池抽真空阀关[SW]
OR D1247.01  ; 复检腔体机构：关闭除破真空阀以外全部阀门（复位）
ANDLD
DIFU(013) 317.08  ; 复测电池抽真空阀关[Pls]
LD TR0
LD 317.08  ; 复测电池抽真空阀关[Pls]
OR 417.08  ; 复测电池抽真空阀关[M]
ANDLD
ANDNOT 309.08  ; 复测电池抽真空阀[Pls]
ANDNOT 835.15  ; 复测电池抽真空阀关到位标志[0000.17]
OUT 417.08  ; 复测电池抽真空阀关[M]

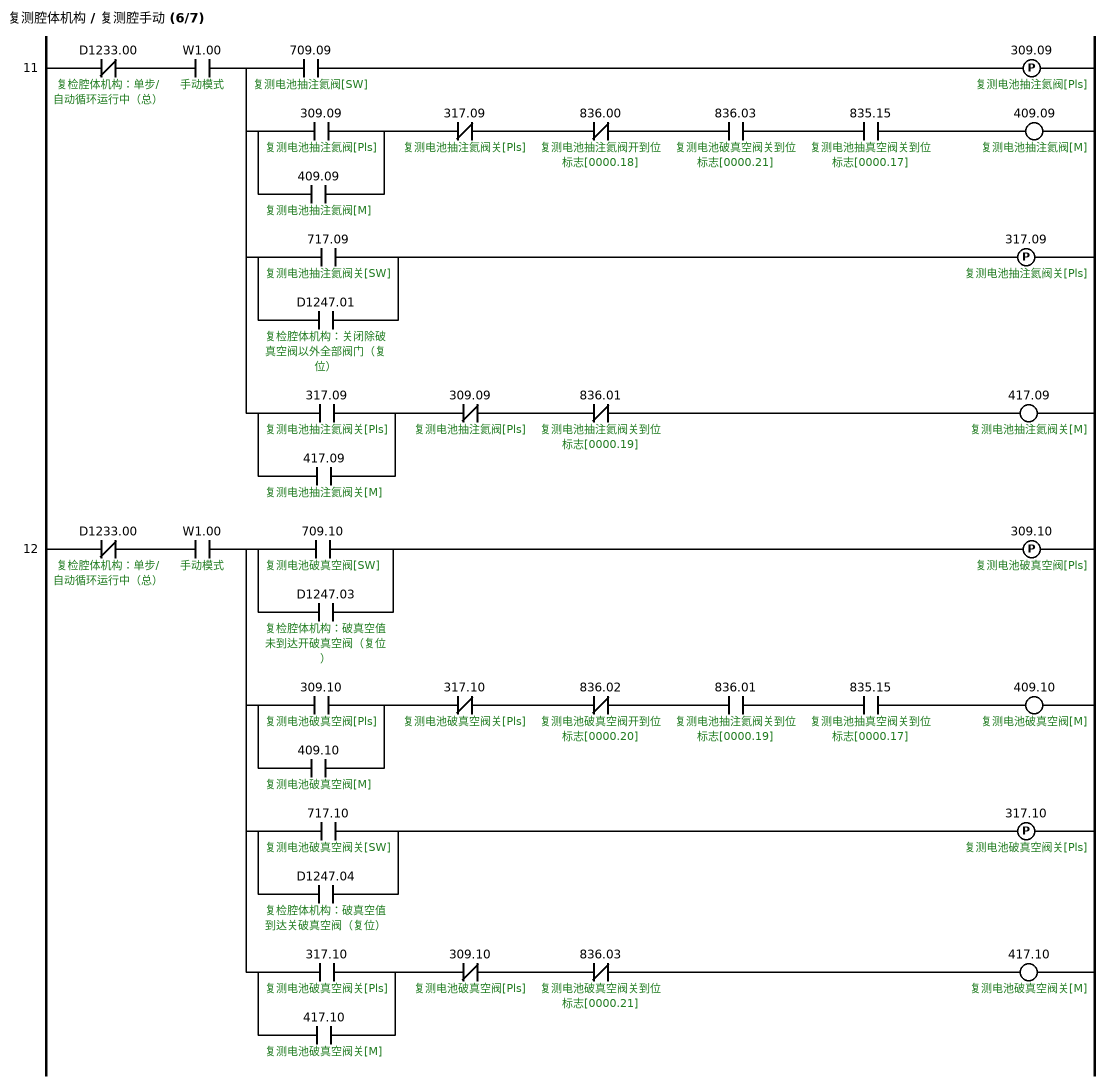
; rung 11
LDNOT D1233.00  ; 复检腔体机构：单步/自动循环运行中（总）
AND W1.00  ; 手动模式
OUT TR0
AND 709.09  ; 复测电池抽注氦阀[SW]
DIFU(013) 309.09  ; 复测电池抽注氦阀[Pls]
LD TR0
LD 309.09  ; 复测电池抽注氦阀[Pls]
OR 409.09  ; 复测电池抽注氦阀[M]
ANDLD
ANDNOT 317.09  ; 复测电池抽注氦阀关[Pls]
ANDNOT 836.00  ; 复测电池抽注氦阀开到位标志[0000.18]
AND 836.03  ; 复测电池破真空阀关到位标志[0000.21]
AND 835.15  ; 复测电池抽真空阀关到位标志[0000.17]
OUT 409.09  ; 复测电池抽注氦阀[M]
LD TR0
LD 717.09  ; 复测电池抽注氦阀关[SW]
OR D1247.01  ; 复检腔体机构：关闭除破真空阀以外全部阀门（复位）
ANDLD
DIFU(013) 317.09  ; 复测电池抽注氦阀关[Pls]
LD TR0
LD 317.09  ; 复测电池抽注氦阀关[Pls]
OR 417.09  ; 复测电池抽注氦阀关[M]
ANDLD
ANDNOT 309.09  ; 复测电池抽注氦阀[Pls]
ANDNOT 836.01  ; 复测电池抽注氦阀关到位标志[0000.19]
OUT 417.09  ; 复测电池抽注氦阀关[M]
; rung 12
LDNOT D1233.00  ; 复检腔体机构：单步/自动循环运行中（总）
AND W1.00  ; 手动模式
OUT TR0
LD 709.10  ; 复测电池破真空阀[SW]
OR D1247.03  ; 复检腔体机构：破真空值未到达开破真空阀（复位）
ANDLD
DIFU(013) 309.10  ; 复测电池破真空阀[Pls]
LD TR0
LD 309.10  ; 复测电池破真空阀[Pls]
OR 409.10  ; 复测电池破真空阀[M]
ANDLD
ANDNOT 317.10  ; 复测电池破真空阀关[Pls]
ANDNOT 836.02  ; 复测电池破真空阀开到位标志[0000.20]
AND 836.01  ; 复测电池抽注氦阀关到位标志[0000.19]
AND 835.15  ; 复测电池抽真空阀关到位标志[0000.17]
OUT 409.10  ; 复测电池破真空阀[M]
LD TR0
LD 717.10  ; 复测电池破真空阀关[SW]
OR D1247.04  ; 复检腔体机构：破真空值到达关破真空阀（复位）
ANDLD
DIFU(013) 317.10  ; 复测电池破真空阀关[Pls]
LD TR0
LD 317.10  ; 复测电池破真空阀关[Pls]
OR 417.10  ; 复测电池破真空阀关[M]
ANDLD
ANDNOT 309.10  ; 复测电池破真空阀[Pls]
ANDNOT 836.03  ; 复测电池破真空阀关到位标志[0000.21]
OUT 417.10  ; 复测电池破真空阀关[M]

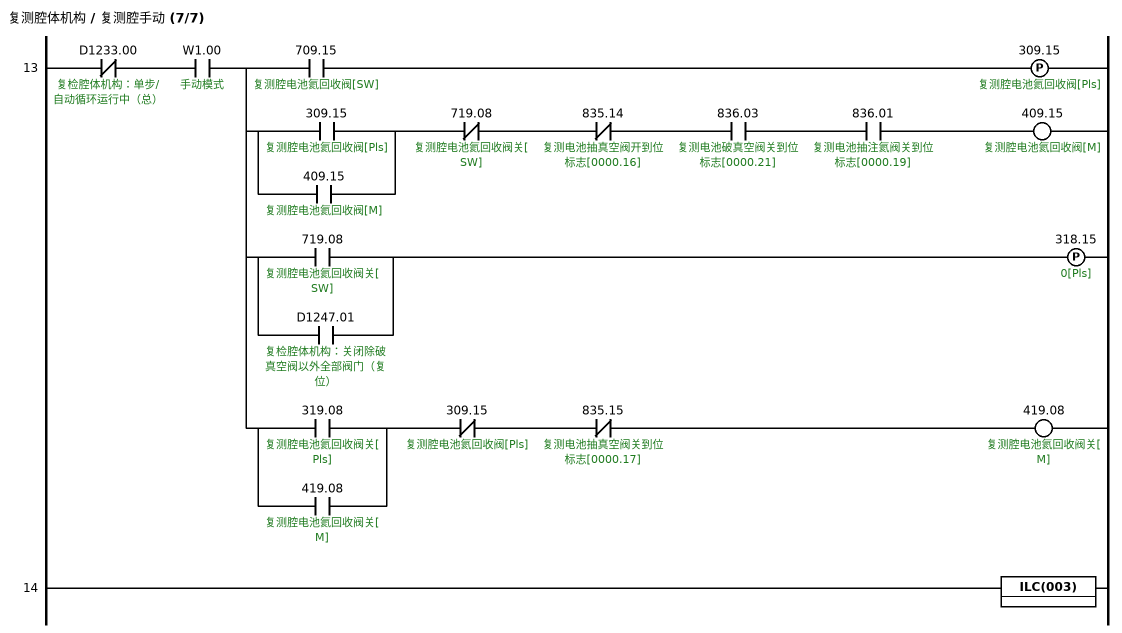
; rung 13
LDNOT D1233.00  ; 复检腔体机构：单步/自动循环运行中（总）
AND W1.00  ; 手动模式
OUT TR0
AND 709.15  ; 复测腔电池氦回收阀[SW]
DIFU(013) 309.15  ; 复测腔电池氦回收阀[Pls]
LD TR0
LD 309.15  ; 复测腔电池氦回收阀[Pls]
OR 409.15  ; 复测腔电池氦回收阀[M]
ANDLD
ANDNOT 719.08  ; 复测腔电池氦回收阀关[SW]
ANDNOT 835.14  ; 复测电池抽真空阀开到位标志[0000.16]
AND 836.03  ; 复测电池破真空阀关到位标志[0000.21]
AND 836.01  ; 复测电池抽注氦阀关到位标志[0000.19]
OUT 409.15  ; 复测腔电池氦回收阀[M]
LD TR0
LD 719.08  ; 复测腔电池氦回收阀关[SW]
OR D1247.01  ; 复检腔体机构：关闭除破真空阀以外全部阀门（复位）
ANDLD
DIFU(013) 318.15  ; 0[Pls]
LD TR0
LD 319.08  ; 复测腔电池氦回收阀关[Pls]
OR 419.08  ; 复测腔电池氦回收阀关[M]
ANDLD
ANDNOT 309.15  ; 复测腔电池氦回收阀[Pls]
ANDNOT 835.15  ; 复测电池抽真空阀关到位标志[0000.17]
OUT 419.08  ; 复测腔电池氦回收阀关[M]
; rung 14
ILC(003)

### Section 复检腔自检

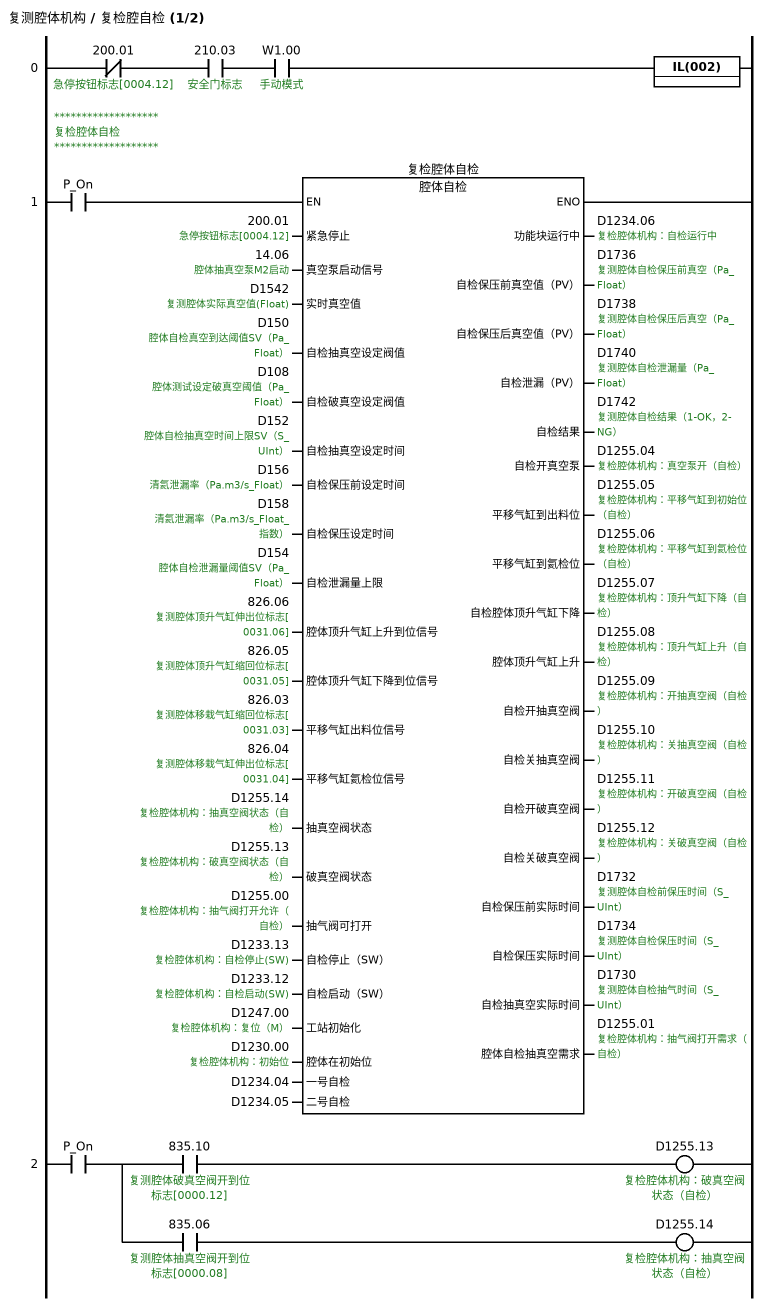
; rung 0
LDNOT 200.01  ; 急停按钮标志[0004.12]
AND 210.03  ; 安全门标志
AND W1.00  ; 手动模式
IL(002)
; rung 1: ******************* / 复检腔体自检 / *******************
LD P_On
CALL 复检腔体自检 : 腔体自检 (紧急停止 := 200.01, 真空泵启动信号 := 14.06, 实时真空值 := D1542, 自检抽真空设定阀值 := D150, 自检破真空设定阀值 := D108, 自检抽真空设定时间 := D152, 自检保压前设定时间 := D156, 自检保压设定时间 := D158, 自检泄漏量上限 := D154, 腔体顶升气缸上升到位信号 := 826.06, 腔体顶升气缸下降到位信号 := 826.05, 平移气缸出料位信号 := 826.03, 平移气缸氦检位信号 := 826.04, 抽真空阀状态 := D1255.14, 破真空阀状态 := D1255.13, 抽气阀可打开 := D1255.00, 自检停止（SW） := D1233.13, 自检启动（SW） := D1233.12, 工站初始化 := D1247.00, 腔体在初始位 := D1230.00, 一号自检 := D1234.04, 二号自检 := D1234.05, 功能块运行中 => D1234.06, 自检保压前真空值（PV） => D1736, 自检保压后真空值（PV） => D1738, 自检泄漏（PV） => D1740, 自检结果 => D1742, 自检开真空泵 => D1255.04, 平移气缸到出料位 => D1255.05, 平移气缸到氦检位 => D1255.06, 自检腔体顶升气缸下降 => D1255.07, 腔体顶升气缸上升 => D1255.08, 自检开抽真空阀 => D1255.09, 自检关抽真空阀 => D1255.10, 自检开破真空阀 => D1255.11, 自检关破真空阀 => D1255.12, 自检保压前实际时间 => D1732, 自检保压实际时间 => D1734, 自检抽真空实际时间 => D1730, 腔体自检抽真空需求 => D1255.01)  ; 急停按钮标志[0004.12], 腔体抽真空泵M2启动, 复测腔体实际真空值(Float), 腔体自检真空到达阈值SV（Pa_Float）, 腔体测试设定破真空阈值（Pa_Float）, 腔体自检抽真空时间上限SV（S_UInt）, 清氦泄漏率（Pa.m3/s_Float）, 清氦泄漏率（Pa.m3/s_Float_指数）, 腔体自检泄漏量阈值SV（Pa_Float）, 复测腔体顶升气缸伸出位标志[0031.06], 复测腔体顶升气缸缩回位标志[0031.05], 复测腔体移栽气缸缩回位标志[0031.03], 复测腔体移栽气缸伸出位标志[0031.04], 复检腔体机构：抽真空阀状态（自检）, 复检腔体机构：破真空阀状态（自检）, 复检腔体机构：抽气阀打开允许（自检）, 复检腔体机构：自检停止(SW), 复检腔体机构：自检启动(SW), 复检腔体机构：复位（M）, 复检腔体机构：初始位, 复检腔体机构：自检运行中, 复测腔体自检保压前真空（Pa_Float）, 复测腔体自检保压后真空（Pa_Float）, 复测腔体自检泄漏量（Pa_Float）, 复测腔体自检结果（1-OK，2-NG）, 复检腔体机构：真空泵开（自检）, 复检腔体机构：平移气缸到初始位（自检）, 复检腔体机构：平移气缸到氦检位（自检）, 复检腔体机构：顶升气缸下降（自检）, 复检腔体机构：顶升气缸上升（自检）, 复检腔体机构：开抽真空阀（自检）, 复检腔体机构：关抽真空阀（自检）, 复检腔体机构：开破真空阀（自检）, 复检腔体机构：关破真空阀（自检）, 复测腔体自检前保压时间（S_UInt）, 复测腔体自检保压时间（S_UInt）, 复测腔体自检抽气时间（S_UInt）, 复检腔体机构：抽气阀打开需求（自检）
; rung 2
LD P_On
OUT TR0
AND 835.10  ; 复测腔体破真空阀开到位标志[0000.12]
OUT D1255.13  ; 复检腔体机构：破真空阀状态（自检）
LD TR0
AND 835.06  ; 复测腔体抽真空阀开到位标志[0000.08]
OUT D1255.14  ; 复检腔体机构：抽真空阀状态（自检）

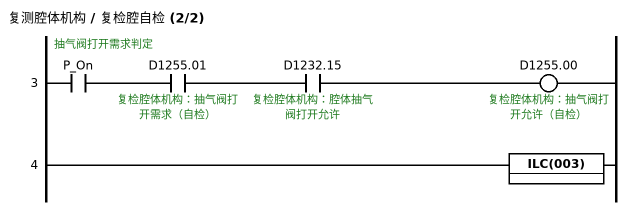
; rung 3: 抽气阀打开需求判定
LD P_On
AND D1255.01  ; 复检腔体机构：抽气阀打开需求（自检）
AND D1232.15  ; 复检腔体机构：腔体抽气阀打开允许
OUT D1255.00  ; 复检腔体机构：抽气阀打开允许（自检）
; rung 4
ILC(003)

### Section 工站复位

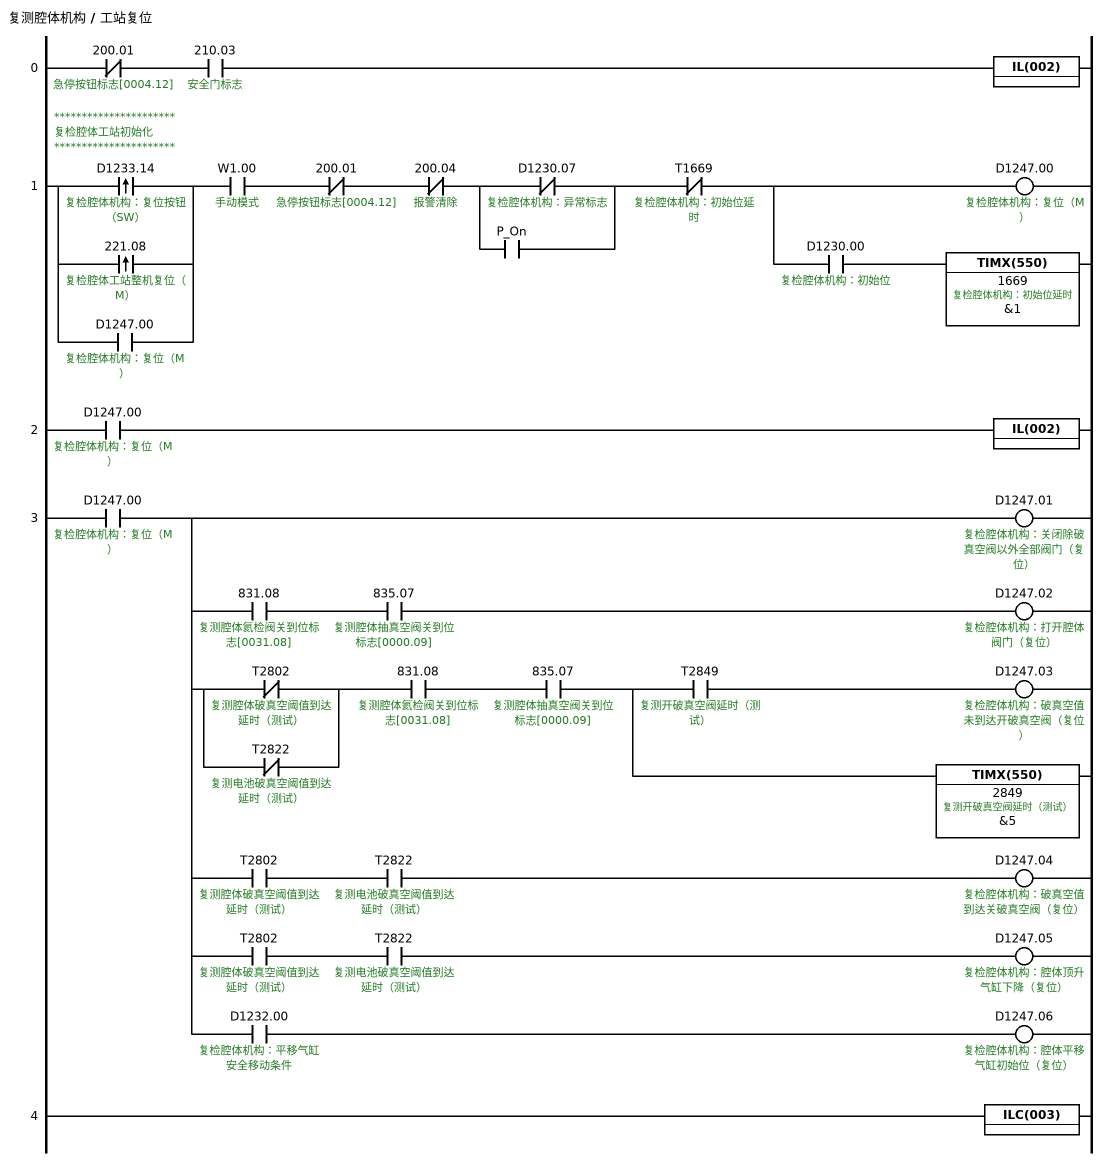
; rung 0
LDNOT 200.01  ; 急停按钮标志[0004.12]
AND 210.03  ; 安全门标志
IL(002)
; rung 1: ********************** / 复检腔体工站初始化 / **********************
@LD D1233.14  ; 复检腔体机构：复位按钮（SW）
@OR 221.08  ; 复检腔体工站整机复位（M）
OR D1247.00  ; 复检腔体机构：复位（M）
AND W1.00  ; 手动模式
ANDNOT 200.01  ; 急停按钮标志[0004.12]
ANDNOT 200.04  ; 报警清除
LDNOT D1230.07  ; 复检腔体机构：异常标志
OR P_On
ANDLD
ANDNOT T1669  ; 复检腔体机构：初始位延时
OUT D1247.00  ; 复检腔体机构：复位（M）
AND D1230.00  ; 复检腔体机构：初始位
TIMX(550) 1669 &1  ; 复检腔体机构：初始位延时
; rung 2
LD D1247.00  ; 复检腔体机构：复位（M）
IL(002)
; rung 3
LD D1247.00  ; 复检腔体机构：复位（M）
OUT TR0
OUT D1247.01  ; 复检腔体机构：关闭除破真空阀以外全部阀门（复位）
AND 831.08  ; 复测腔体氦检阀关到位标志[0031.08]
AND 835.07  ; 复测腔体抽真空阀关到位标志[0000.09]
OUT D1247.02  ; 复检腔体机构：打开腔体阀门（复位）
LD TR0
LDNOT T2802  ; 复测腔体破真空阈值到达延时（测试）
ORNOT T2822  ; 复测电池破真空阈值到达延时（测试）
ANDLD
AND 831.08  ; 复测腔体氦检阀关到位标志[0031.08]
AND 835.07  ; 复测腔体抽真空阀关到位标志[0000.09]
OUT TR1
AND T2849  ; 复测开破真空阀延时（测试）
OUT D1247.03  ; 复检腔体机构：破真空值未到达开破真空阀（复位）
LD TR1
TIMX(550) 2849 &5  ; 复测开破真空阀延时（测试）
LD TR0
AND T2802  ; 复测腔体破真空阈值到达延时（测试）
AND T2822  ; 复测电池破真空阈值到达延时（测试）
OUT D1247.04  ; 复检腔体机构：破真空值到达关破真空阀（复位）
LD TR0
AND T2802  ; 复测腔体破真空阈值到达延时（测试）
AND T2822  ; 复测电池破真空阈值到达延时（测试）
OUT D1247.05  ; 复检腔体机构：腔体顶升气缸下降（复位）
LD TR0
AND D1232.00  ; 复检腔体机构：平移气缸安全移动条件
OUT D1247.06  ; 复检腔体机构：腔体平移气缸初始位（复位）
; rung 4
ILC(003)

### Section 指示灯

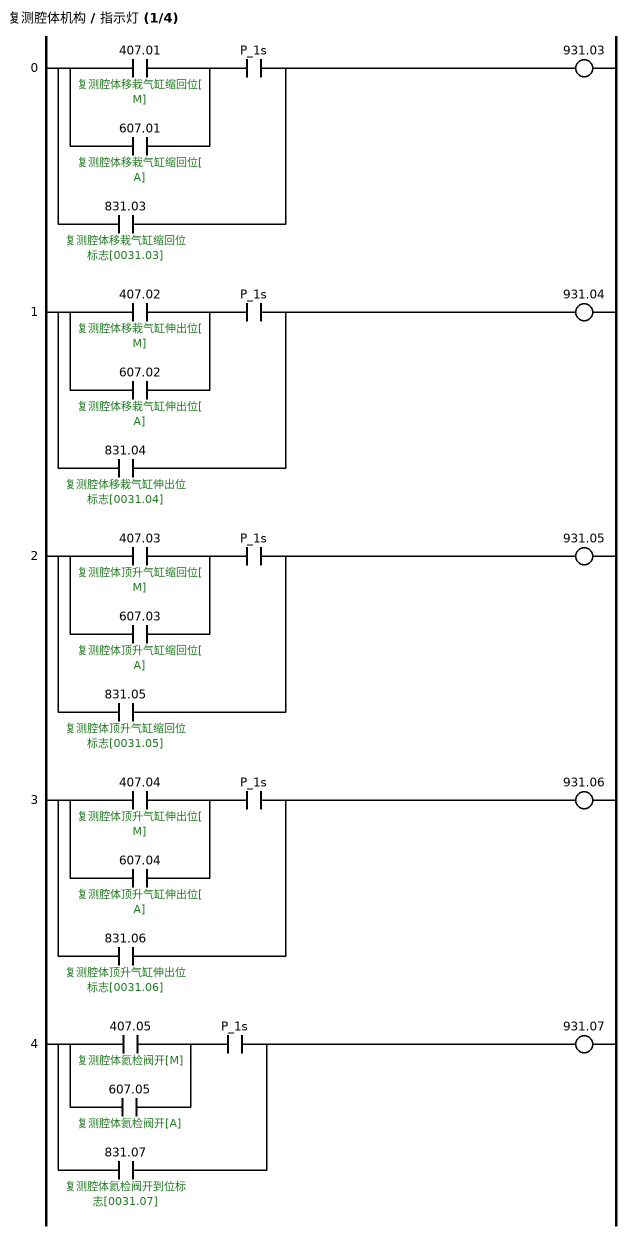
; rung 0
LD 407.01  ; 复测腔体移栽气缸缩回位[M]
OR 607.01  ; 复测腔体移栽气缸缩回位[A]
AND P_1s
OR 831.03  ; 复测腔体移栽气缸缩回位标志[0031.03]
OUT 931.03
; rung 1
LD 407.02  ; 复测腔体移栽气缸伸出位[M]
OR 607.02  ; 复测腔体移栽气缸伸出位[A]
AND P_1s
OR 831.04  ; 复测腔体移栽气缸伸出位标志[0031.04]
OUT 931.04
; rung 2
LD 407.03  ; 复测腔体顶升气缸缩回位[M]
OR 607.03  ; 复测腔体顶升气缸缩回位[A]
AND P_1s
OR 831.05  ; 复测腔体顶升气缸缩回位标志[0031.05]
OUT 931.05
; rung 3
LD 407.04  ; 复测腔体顶升气缸伸出位[M]
OR 607.04  ; 复测腔体顶升气缸伸出位[A]
AND P_1s
OR 831.06  ; 复测腔体顶升气缸伸出位标志[0031.06]
OUT 931.06
; rung 4
LD 407.05  ; 复测腔体氦检阀开[M]
OR 607.05  ; 复测腔体氦检阀开[A]
AND P_1s
OR 831.07  ; 复测腔体氦检阀开到位标志[0031.07]
OUT 931.07

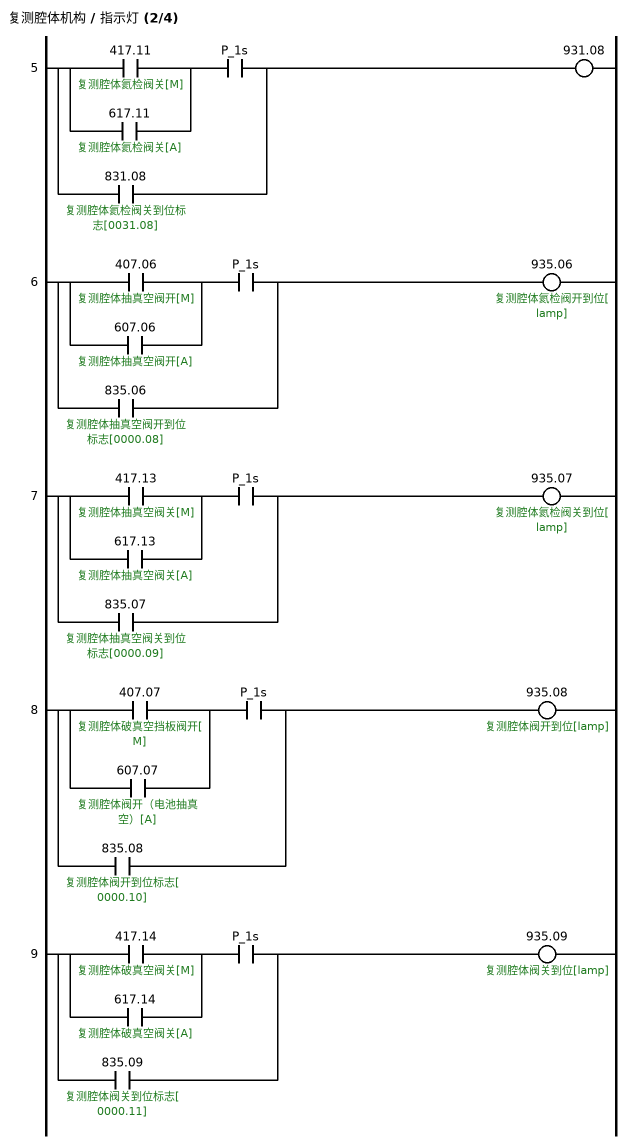
; rung 5
LD 417.11  ; 复测腔体氦检阀关[M]
OR 617.11  ; 复测腔体氦检阀关[A]
AND P_1s
OR 831.08  ; 复测腔体氦检阀关到位标志[0031.08]
OUT 931.08
; rung 6
LD 407.06  ; 复测腔体抽真空阀开[M]
OR 607.06  ; 复测腔体抽真空阀开[A]
AND P_1s
OR 835.06  ; 复测腔体抽真空阀开到位标志[0000.08]
OUT 935.06  ; 复测腔体氦检阀开到位[lamp]
; rung 7
LD 417.13  ; 复测腔体抽真空阀关[M]
OR 617.13  ; 复测腔体抽真空阀关[A]
AND P_1s
OR 835.07  ; 复测腔体抽真空阀关到位标志[0000.09]
OUT 935.07  ; 复测腔体氦检阀关到位[lamp]
; rung 8
LD 407.07  ; 复测腔体破真空挡板阀开[M]
OR 607.07  ; 复测腔体阀开（电池抽真空）[A]
AND P_1s
OR 835.08  ; 复测腔体阀开到位标志[0000.10]
OUT 935.08  ; 复测腔体阀开到位[lamp]
; rung 9
LD 417.14  ; 复测腔体破真空阀关[M]
OR 617.14  ; 复测腔体破真空阀关[A]
AND P_1s
OR 835.09  ; 复测腔体阀关到位标志[0000.11]
OUT 935.09  ; 复测腔体阀关到位[lamp]

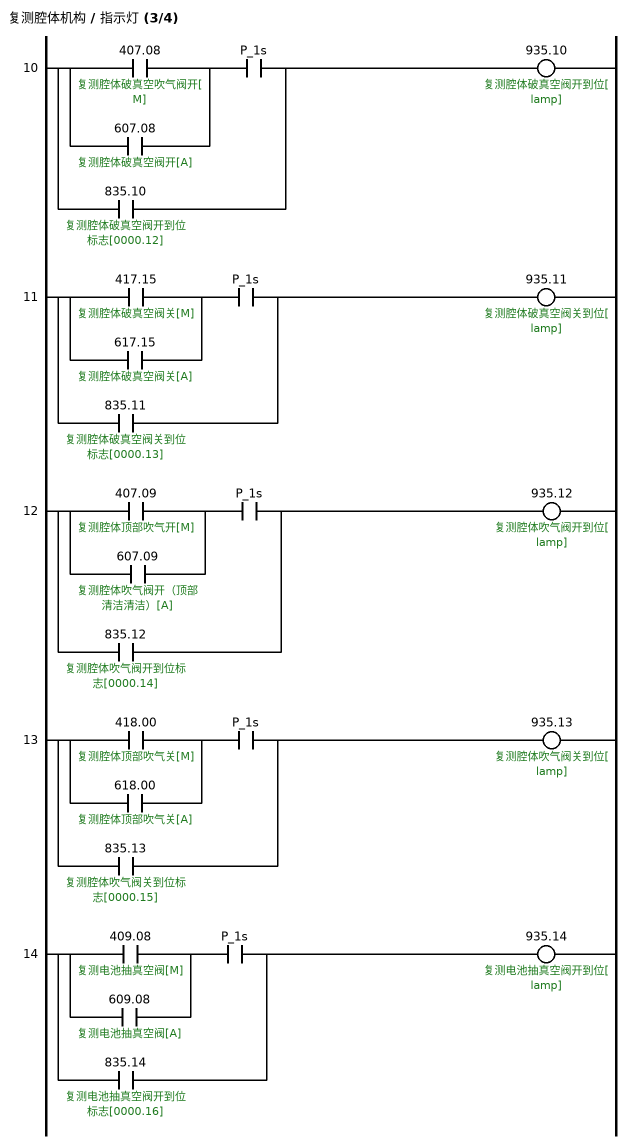
; rung 10
LD 407.08  ; 复测腔体破真空吹气阀开[M]
OR 607.08  ; 复测腔体破真空阀开[A]
AND P_1s
OR 835.10  ; 复测腔体破真空阀开到位标志[0000.12]
OUT 935.10  ; 复测腔体破真空阀开到位[lamp]
; rung 11
LD 417.15  ; 复测腔体破真空阀关[M]
OR 617.15  ; 复测腔体破真空阀关[A]
AND P_1s
OR 835.11  ; 复测腔体破真空阀关到位标志[0000.13]
OUT 935.11  ; 复测腔体破真空阀关到位[lamp]
; rung 12
LD 407.09  ; 复测腔体顶部吹气开[M]
OR 607.09  ; 复测腔体吹气阀开（顶部清洁清洁）[A]
AND P_1s
OR 835.12  ; 复测腔体吹气阀开到位标志[0000.14]
OUT 935.12  ; 复测腔体吹气阀开到位[lamp]
; rung 13
LD 418.00  ; 复测腔体顶部吹气关[M]
OR 618.00  ; 复测腔体顶部吹气关[A]
AND P_1s
OR 835.13  ; 复测腔体吹气阀关到位标志[0000.15]
OUT 935.13  ; 复测腔体吹气阀关到位[lamp]
; rung 14
LD 409.08  ; 复测电池抽真空阀[M]
OR 609.08  ; 复测电池抽真空阀[A]
AND P_1s
OR 835.14  ; 复测电池抽真空阀开到位标志[0000.16]
OUT 935.14  ; 复测电池抽真空阀开到位[lamp]

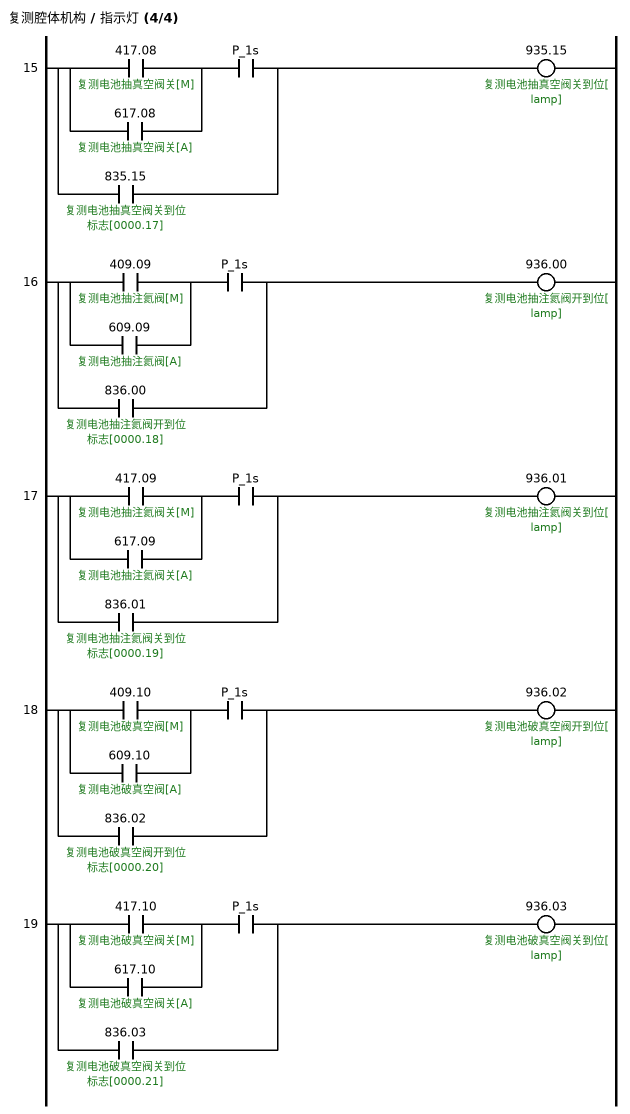
; rung 15
LD 417.08  ; 复测电池抽真空阀关[M]
OR 617.08  ; 复测电池抽真空阀关[A]
AND P_1s
OR 835.15  ; 复测电池抽真空阀关到位标志[0000.17]
OUT 935.15  ; 复测电池抽真空阀关到位[lamp]
; rung 16
LD 409.09  ; 复测电池抽注氦阀[M]
OR 609.09  ; 复测电池抽注氦阀[A]
AND P_1s
OR 836.00  ; 复测电池抽注氦阀开到位标志[0000.18]
OUT 936.00  ; 复测电池抽注氦阀开到位[lamp]
; rung 17
LD 417.09  ; 复测电池抽注氦阀关[M]
OR 617.09  ; 复测电池抽注氦阀关[A]
AND P_1s
OR 836.01  ; 复测电池抽注氦阀关到位标志[0000.19]
OUT 936.01  ; 复测电池抽注氦阀关到位[lamp]
; rung 18
LD 409.10  ; 复测电池破真空阀[M]
OR 609.10  ; 复测电池破真空阀[A]
AND P_1s
OR 836.02  ; 复测电池破真空阀开到位标志[0000.20]
OUT 936.02  ; 复测电池破真空阀开到位[lamp]
; rung 19
LD 417.10  ; 复测电池破真空阀关[M]
OR 617.10  ; 复测电池破真空阀关[A]
AND P_1s
OR 836.03  ; 复测电池破真空阀关到位标志[0000.21]
OUT 936.03  ; 复测电池破真空阀关到位[lamp]

### Section 外部输出

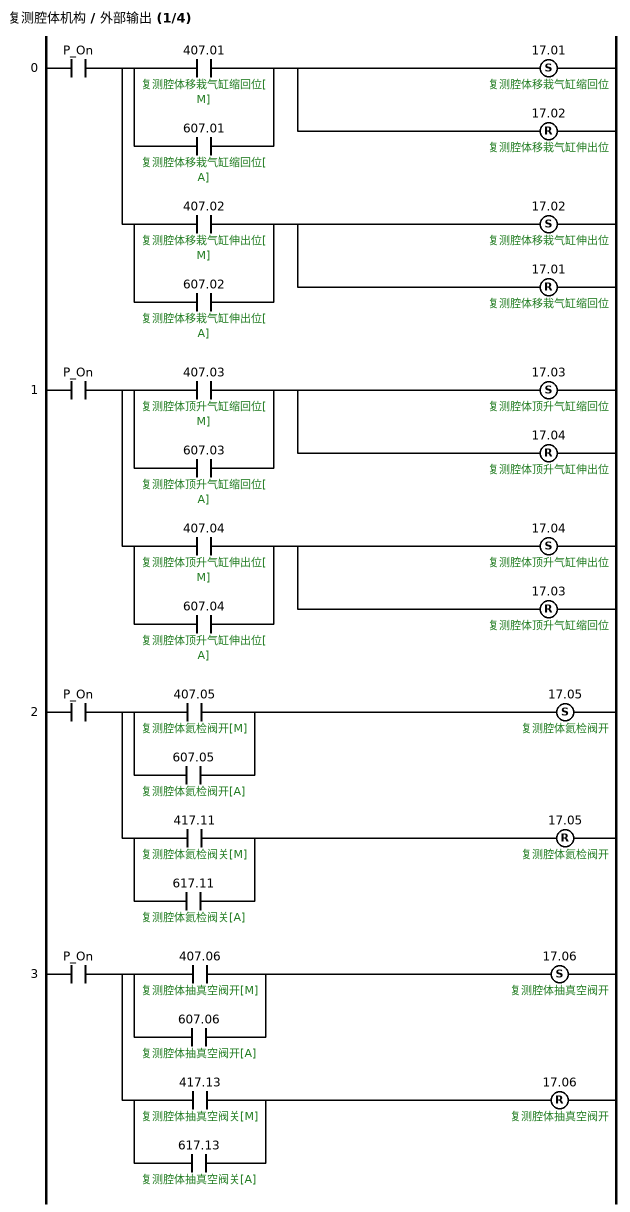
; rung 0
LD P_On
OUT TR0
LD 407.01  ; 复测腔体移栽气缸缩回位[M]
OR 607.01  ; 复测腔体移栽气缸缩回位[A]
ANDLD
SET 17.01  ; 复测腔体移栽气缸缩回位
RSET 17.02  ; 复测腔体移栽气缸伸出位
LD TR0
LD 407.02  ; 复测腔体移栽气缸伸出位[M]
OR 607.02  ; 复测腔体移栽气缸伸出位[A]
ANDLD
SET 17.02  ; 复测腔体移栽气缸伸出位
RSET 17.01  ; 复测腔体移栽气缸缩回位
; rung 1
LD P_On
OUT TR0
LD 407.03  ; 复测腔体顶升气缸缩回位[M]
OR 607.03  ; 复测腔体顶升气缸缩回位[A]
ANDLD
SET 17.03  ; 复测腔体顶升气缸缩回位
RSET 17.04  ; 复测腔体顶升气缸伸出位
LD TR0
LD 407.04  ; 复测腔体顶升气缸伸出位[M]
OR 607.04  ; 复测腔体顶升气缸伸出位[A]
ANDLD
SET 17.04  ; 复测腔体顶升气缸伸出位
RSET 17.03  ; 复测腔体顶升气缸缩回位
; rung 2
LD P_On
OUT TR0
LD 407.05  ; 复测腔体氦检阀开[M]
OR 607.05  ; 复测腔体氦检阀开[A]
ANDLD
SET 17.05  ; 复测腔体氦检阀开
LD TR0
LD 417.11  ; 复测腔体氦检阀关[M]
OR 617.11  ; 复测腔体氦检阀关[A]
ANDLD
RSET 17.05  ; 复测腔体氦检阀开
; rung 3
LD P_On
OUT TR0
LD 407.06  ; 复测腔体抽真空阀开[M]
OR 607.06  ; 复测腔体抽真空阀开[A]
ANDLD
SET 17.06  ; 复测腔体抽真空阀开
LD TR0
LD 417.13  ; 复测腔体抽真空阀关[M]
OR 617.13  ; 复测腔体抽真空阀关[A]
ANDLD
RSET 17.06  ; 复测腔体抽真空阀开

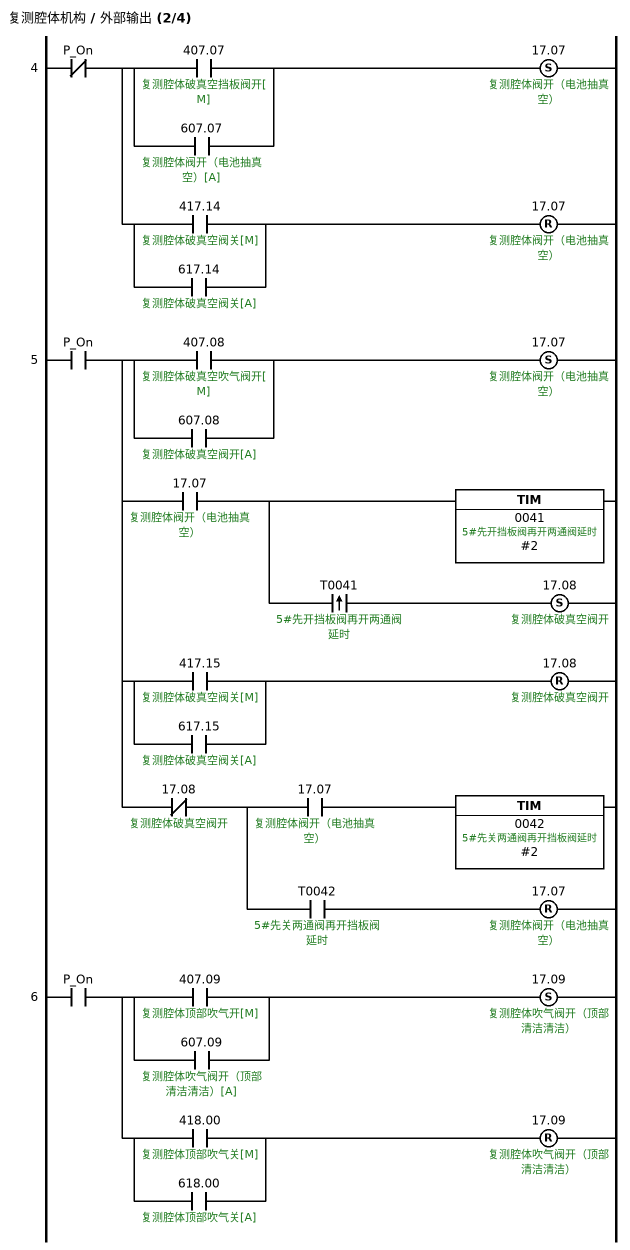
; rung 4
LDNOT P_On
OUT TR0
LD 407.07  ; 复测腔体破真空挡板阀开[M]
OR 607.07  ; 复测腔体阀开（电池抽真空）[A]
ANDLD
SET 17.07  ; 复测腔体阀开（电池抽真空）
LD TR0
LD 417.14  ; 复测腔体破真空阀关[M]
OR 617.14  ; 复测腔体破真空阀关[A]
ANDLD
RSET 17.07  ; 复测腔体阀开（电池抽真空）
; rung 5
LD P_On
OUT TR0
LD 407.08  ; 复测腔体破真空吹气阀开[M]
OR 607.08  ; 复测腔体破真空阀开[A]
ANDLD
SET 17.07  ; 复测腔体阀开（电池抽真空）
LD TR0
AND 17.07  ; 复测腔体阀开（电池抽真空）
TIM 0041 #2  ; 5#先开挡板阀再开两通阀延时
@AND T0041  ; 5#先开挡板阀再开两通阀延时
SET 17.08  ; 复测腔体破真空阀开
LD TR0
LD 417.15  ; 复测腔体破真空阀关[M]
OR 617.15  ; 复测腔体破真空阀关[A]
ANDLD
RSET 17.08  ; 复测腔体破真空阀开
LD TR0
ANDNOT 17.08  ; 复测腔体破真空阀开
OUT TR0
AND 17.07  ; 复测腔体阀开（电池抽真空）
TIM 0042 #2  ; 5#先关两通阀再开挡板阀延时
LD TR0
AND T0042  ; 5#先关两通阀再开挡板阀延时
RSET 17.07  ; 复测腔体阀开（电池抽真空）
; rung 6
LD P_On
OUT TR0
LD 407.09  ; 复测腔体顶部吹气开[M]
OR 607.09  ; 复测腔体吹气阀开（顶部清洁清洁）[A]
ANDLD
SET 17.09  ; 复测腔体吹气阀开（顶部清洁清洁）
LD TR0
LD 418.00  ; 复测腔体顶部吹气关[M]
OR 618.00  ; 复测腔体顶部吹气关[A]
ANDLD
RSET 17.09  ; 复测腔体吹气阀开（顶部清洁清洁）

